C01784=1018.321,266.101,-148.009,-25.446,21.246,-34.279
C01785=1018.328,265.821,-147.958,-25.406,21.239,-34.538
C01786=1018.334,265.575,-147.912,-25.370,21.233,-34.766
C01787=1018.341,265.330,-147.868,-25.335,21.229,-34.991
C01788=1018.347,265.084,-147.824,-25.300,21.225,-35.219
C01789=1018.352,264.837,-147.781,-25.265,21.221,-35.444
C01790=1018.357,264.558,-147.733,-25.226,21.219,-35.699
C01791=1018.363,264.279,-147.684,-25.186,21.217,-35.952
C01792=1018.367,264.000,-147.637,-25.147,21.216,-36.205
C01793=1018.371,263.721,-147.591,-25.108,21.215,-36.458
C01794=1018.374,263.474,-147.551,-25.074,21.216,-36.681
C01795=1018.377,263.227,-147.511,-25.040,21.217,-36.903
C01796=1018.379,262.980,-147.472,-25.006,21.220,-37.124
C01797=1018.382,262.733,-147.433,-24.973,21.223,-37.345
C01798=1018.384,262.453,-147.389,-24.935,21.227,-37.593
C01799=1018.386,262.174,-147.346,-24.897,21.233,-37.842
C01800=1018.387,261.895,-147.304,-24.860,21.238,-38.090
C01801=1018.387,261.616,-147.262,-24.823,21.245,-38.337
C01802=1018.388,261.368,-147.227,-24.790,21.251,-38.554
C01803=1018.388,261.121,-147.191,-24.758,21.259,-38.770
C01804=1018.388,260.874,-147.156,-24.725,21.267,-38.988
C01805=1018.386,260.625,-147.121,-24.693,21.275,-39.204
C01806=1018.385,260.346,-147.083,-24.658,21.287,-39.446
C01807=1018.383,260.066,-147.044,-24.622,21.298,-39.688
C01808=1018.381,259.787,-147.008,-24.587,21.310,-39.930
C01809=1018.378,259.507,-146.971,-24.551,21.322,-40.171
C01810=1018.361,258.272,-146.818,-24.430,21.375,-41.012
C01811=1018.358,258.028,-146.788,-24.430,21.375,-41.014
C01812=1018.355,257.784,-146.759,-24.429,21.375,-41.018
C01813=1018.351,257.541,-146.731,-24.429,21.376,-41.019
C01814=1018.347,257.298,-146.701,-24.429,21.376,-41.021
C01815=1018.344,257.054,-146.671,-24.428,21.375,-41.025
C01816=1018.341,256.811,-146.642,-24.428,21.376,-41.027
C01817=1018.337,256.567,-146.614,-24.428,21.377,-41.029
C01818=1018.334,256.318,-146.584,-24.427,21.376,-41.032
C01819=1018.331,256.071,-146.554,-24.427,21.376,-41.034
C01820=1018.327,255.822,-146.525,-24.426,21.376,-41.037
C01821=1018.323,255.574,-146.495,-24.426,21.377,-41.040
C01822=1018.321,255.326,-146.465,-24.426,21.377,-41.042
C01823=1018.317,255.078,-146.435,-24.425,21.377,-41.045
C01824=1018.314,254.829,-146.406,-24.425,21.377,-41.047
C01825=1018.310,254.581,-146.376,-24.425,21.377,-41.049
C01826=1018.307,254.333,-146.347,-24.424,21.378,-41.052
C01827=1018.303,254.084,-146.318,-24.424,21.378,-41.054
C01828=1018.300,253.837,-146.288,-24.424,21.378,-41.058
C01829=1018.297,253.588,-146.258,-24.423,21.378,-41.060
C01830=1018.293,253.341,-146.229,-24.423,21.378,-41.061
C01831=1018.290,253.092,-146.199,-24.423,21.378,-41.065
C01832=1018.287,252.844,-146.170,-24.422,21.379,-41.067
C01833=1018.283,252.595,-146.140,-24.422,21.379,-41.069
C01834=1018.280,252.347,-146.111,-24.421,21.378,-41.072
C01835=1018.277,252.098,-146.081,-24.421,21.379,-41.074
C01836=1018.274,251.850,-146.053,-24.421,21.380,-41.076
C01837=1018.270,251.602,-146.022,-24.421,21.380,-41.078
C01838=1018.267,251.359,-145.994,-24.420,21.380,-41.082
C01839=1018.264,251.116,-145.965,-24.420,21.380,-41.084
C01840=1018.260,250.872,-145.937,-24.420,21.380,-41.085
C01841=1018.258,250.629,-145.908,-24.419,21.380,-41.089
C01842=1018.255,250.385,-145.879,-24.419,21.380,-41.091
C01843=1018.251,250.142,-145.850,-24.419,21.381,-41.093
C01844=1018.248,249.899,-145.821,-24.418,21.381,-41.095
C01845=1018.244,249.656,-145.793,-24.418,21.381,-41.098
C01846=1018.242,249.408,-145.763,-24.418,21.381,-41.100
C01847=1018.238,249.159,-145.734,-24.417,21.381,-41.102
C01848=1018.235,248.911,-145.705,-24.417,21.381,-41.104
C01849=1018.232,248.663,-145.676,-24.417,21.381,-41.107
C01850=1018.229,248.414,-145.646,-24.416,21.381,-41.109
C01851=1018.226,248.166,-145.617,-24.416,21.382,-41.111
C01852=1018.222,247.918,-145.588,-24.416,21.382,-41.113
C01853=1018.219,247.669,-145.558,-24.415,21.382,-41.117
C01854=1018.216,247.421,-145.529,-24.415,21.382,-41.118
C01855=1018.213,247.173,-145.500,-24.415,21.382,-41.120
C01856=1018.210,246.925,-145.471,-24.414,21.383,-41.122
C01857=1018.207,246.676,-145.441,-24.414,21.382,-41.126
C01858=1018.204,246.428,-145.413,-24.414,21.382,-41.127
C01859=1018.200,246.180,-145.384,-24.413,21.383,-41.129
C01860=1018.198,245.932,-145.354,-24.413,21.384,-41.132
C01861=1018.194,245.683,-145.325,-24.413,21.384,-41.134
C01862=1018.191,245.435,-145.296,-24.412,21.384,-41.137
C01863=1018.188,245.187,-145.267,-24.412,21.384,-41.139
C01864=1018.185,244.939,-145.238,-24.412,21.384,-41.141
C01865=1018.182,244.690,-145.209,-24.412,21.384,-41.143
C01866=1018.179,244.447,-145.181,-24.411,21.384,-41.144
C01867=1018.176,244.204,-145.152,-24.411,21.384,-41.148
C01868=1018.172,243.961,-145.124,-24.411,21.384,-41.150
C01869=1018.170,243.717,-145.095,-24.410,21.384,-41.151
C01870=1018.167,243.474,-145.067,-24.410,21.385,-41.153
C01871=1018.164,243.231,-145.038,-24.410,21.385,-41.155
C01872=1018.161,242.988,-145.010,-24.410,21.385,-41.157
C01873=1018.158,242.745,-144.981,-24.409,21.385,-41.159
C01874=1018.155,242.497,-144.953,-24.409,21.385,-41.162
C01875=1018.153,242.248,-144.924,-24.408,21.385,-41.164
C01876=1018.149,241.999,-144.895,-24.408,21.385,-41.166
C01877=1018.146,241.751,-144.866,-24.408,21.386,-41.168
C01878=1018.143,241.503,-144.837,-24.408,21.386,-41.170
C01879=1018.140,241.255,-144.808,-24.407,21.386,-41.172
C01880=1018.138,241.006,-144.779,-24.407,21.386,-41.174
C01881=1018.134,240.758,-144.751,-24.407,21.386,-41.177
C01882=1018.132,240.510,-144.721,-24.406,21.386,-41.179
C01883=1018.129,240.262,-144.692,-24.406,21.386,-41.181
C01884=1018.126,240.013,-144.664,-24.406,21.386,-41.183
C01885=1018.123,239.765,-144.635,-24.406,21.387,-41.184
C01886=1018.120,239.517,-144.606,-24.405,21.387,-41.186
C01887=1018.117,239.268,-144.578,-24.405,21.387,-41.188
C01888=1018.114,239.020,-144.549,-24.405,21.387,-41.190
C01889=1018.111,238.772,-144.520,-24.405,21.388,-41.192
C01890=1018.109,238.523,-144.491,-24.404,21.387,-41.195
C01891=1018.106,238.275,-144.462,-24.404,21.387,-41.197
C01892=1018.102,238.027,-144.434,-24.403,21.388,-41.199
C01893=1018.100,237.778,-144.405,-24.403,21.388,-41.201
C01894=1018.096,237.535,-144.376,-24.403,21.388,-41.203
C01895=1018.094,237.291,-144.348,-24.403,21.388,-41.205
C01896=1018.091,237.049,-144.320,-24.402,21.388,-41.207
C01897=1018.088,236.806,-144.292,-24.402,21.389,-41.209
C01898=1018.086,236.562,-144.264,-24.402,21.389,-41.210
C01899=1018.083,236.320,-144.236,-24.402,21.389,-41.212
C01900=1018.081,236.077,-144.208,-24.401,21.389,-41.214
C01901=1018.078,235.833,-144.181,-24.401,21.390,-41.216
C01902=1018.075,235.585,-144.151,-24.401,21.389,-41.218
C01903=1018.072,235.336,-144.123,-24.401,21.389,-41.219
C01904=1018.069,235.089,-144.094,-24.400,21.389,-41.221
C01905=1018.067,234.840,-144.066,-24.400,21.390,-41.223
C01906=1018.064,234.592,-144.037,-24.400,21.390,-41.225
C01907=1018.061,234.343,-144.009,-24.400,21.390,-41.227
C01908=1018.058,234.095,-143.980,-24.399,21.390,-41.229
C01909=1018.055,233.846,-143.951,-24.399,21.390,-41.231
C01910=1018.053,233.598,-143.922,-24.399,21.391,-41.233
C01911=1018.050,233.350,-143.894,-24.399,21.391,-41.234
C01912=1018.047,233.101,-143.866,-24.398,21.391,-41.236
C01913=1018.045,232.853,-143.837,-24.398,21.390,-41.238
C01914=1018.042,232.605,-143.809,-24.398,21.391,-41.240
C01915=1018.039,232.357,-143.780,-24.397,21.391,-41.242
C01916=1018.036,232.108,-143.751,-24.397,21.391,-41.243
C01917=1018.034,231.860,-143.724,-24.397,21.391,-41.245
C01918=1018.031,231.612,-143.694,-24.397,21.392,-41.247
C01919=1018.028,231.363,-143.666,-24.396,21.392,-41.249
C01920=1018.026,231.114,-143.638,-24.396,21.392,-41.251
C01921=1018.023,230.866,-143.609,-24.396,21.391,-41.252
C01922=1018.021,230.624,-143.582,-24.396,21.392,-41.254
C01923=1018.018,230.380,-143.554,-24.395,21.392,-41.256
C01924=1018.015,230.137,-143.526,-24.395,21.392,-41.258
C01925=1018.013,229.894,-143.499,-24.395,21.392,-41.260
C01926=1018.010,229.652,-143.470,-24.395,21.392,-41.262
C01927=1018.008,229.408,-143.442,-24.394,21.392,-41.263
C01928=1018.005,229.166,-143.415,-24.394,21.392,-41.265
C01929=1018.002,228.922,-143.388,-24.394,21.393,-41.266
C01930=1018.000,228.673,-143.359,-24.394,21.393,-41.267
C01931=1017.997,228.426,-143.331,-24.394,21.393,-41.269
C01932=1017.995,228.177,-143.302,-24.393,21.394,-41.271
C01933=1017.992,227.929,-143.274,-24.393,21.393,-41.273
C01934=1017.990,227.681,-143.246,-24.393,21.393,-41.275
C01935=1017.988,227.432,-143.217,-24.393,21.393,-41.276
C01936=1017.985,227.183,-143.189,-24.392,21.394,-41.278
C01937=1017.981,226.935,-143.161,-24.392,21.394,-41.280
C01938=1017.980,226.687,-143.132,-24.392,21.393,-41.282
C01939=1017.977,226.439,-143.104,-24.391,21.393,-41.284
C01940=1017.975,226.190,-143.076,-24.391,21.394,-41.285
C01941=1017.972,225.942,-143.048,-24.391,21.395,-41.286
C01942=1017.969,225.693,-143.020,-24.391,21.395,-41.288
C01943=1017.968,225.445,-142.992,-24.391,21.394,-41.289
C01944=1017.965,225.196,-142.963,-24.390,21.394,-41.291
C01945=1017.962,224.948,-142.935,-24.390,21.395,-41.293
C01946=1017.960,224.700,-142.907,-24.390,21.395,-41.295
C01947=1017.957,224.452,-142.878,-24.390,21.395,-41.297
C01948=1017.954,224.204,-142.851,-24.389,21.394,-41.298
C01949=1017.952,223.955,-142.822,-24.389,21.395,-41.300
C01950=1017.949,223.695,-142.793,-24.389,21.395,-41.300
C01951=1017.948,223.437,-142.764,-24.389,21.396,-41.302
C01952=1017.945,223.177,-142.734,-24.389,21.396,-41.304
C01953=1017.942,222.918,-142.705,-24.388,21.396,-41.306
C01954=1017.940,222.670,-142.677,-24.388,21.395,-41.308
C01955=1017.937,222.421,-142.649,-24.388,21.396,-41.309
C01956=1017.936,222.173,-142.621,-24.388,21.396,-41.311
C01957=1017.933,221.924,-142.593,-24.387,21.396,-41.313
C01958=1017.930,221.676,-142.565,-24.387,21.395,-41.315
C01959=1017.928,221.428,-142.536,-24.387,21.396,-41.315
C01960=1017.925,221.179,-142.508,-24.387,21.397,-41.317
C01961=1017.923,220.931,-142.481,-24.387,21.397,-41.319
C01962=1017.921,220.682,-142.452,-24.386,21.396,-41.320
C01963=1017.918,220.434,-142.424,-24.386,21.396,-41.322
C01964=1017.915,220.186,-142.396,-24.386,21.397,-41.324
C01965=1017.914,219.937,-142.369,-24.386,21.397,-41.325
C01966=1017.912,219.689,-142.341,-24.385,21.397,-41.326
C01967=1017.909,219.440,-142.313,-24.385,21.397,-41.328
C01968=1017.907,219.192,-142.284,-24.385,21.397,-41.330
C01969=1017.904,218.944,-142.256,-24.385,21.397,-41.332
C01970=1017.902,218.695,-142.228,-24.384,21.397,-41.333
C01971=1017.900,218.446,-142.201,-24.384,21.398,-41.333
C01972=1017.897,218.198,-142.173,-24.384,21.398,-41.335
C01973=1017.895,217.949,-142.144,-24.384,21.398,-41.337
C01974=1017.893,217.724,-142.119,-24.384,21.397,-41.339
C01975=1017.891,217.497,-142.094,-24.383,21.398,-41.341
C01976=1017.889,217.270,-142.068,-24.383,21.399,-41.341
C01977=1017.887,217.043,-142.044,-24.383,21.398,-41.342
C01978=1017.885,216.800,-142.016,-24.383,21.398,-41.344
C01979=1017.883,216.558,-141.989,-24.383,21.398,-41.346
C01980=1017.881,216.315,-141.961,-24.383,21.398,-41.346
C01981=1017.878,216.072,-141.934,-24.382,21.399,-41.348
C01982=1017.876,215.829,-141.907,-24.382,21.399,-41.350
C01983=1017.874,215.586,-141.880,-24.382,21.399,-41.352
C01984=1017.872,215.343,-141.852,-24.382,21.398,-41.353
C01985=1017.869,215.101,-141.825,-24.382,21.399,-41.354
C01986=1017.868,214.852,-141.798,-24.381,21.400,-41.356
C01987=1017.865,214.604,-141.770,-24.381,21.399,-41.357
C01988=1017.863,214.356,-141.742,-24.381,21.399,-41.359
C01989=1017.861,214.107,-141.714,-24.381,21.400,-41.359
C01990=1017.859,213.859,-141.687,-24.381,21.400,-41.361
C01991=1017.857,213.610,-141.658,-24.380,21.400,-41.363
C01992=1017.855,213.362,-141.631,-24.380,21.400,-41.365
C01993=1017.852,213.114,-141.603,-24.380,21.400,-41.366
C01994=1017.851,212.865,-141.576,-24.380,21.400,-41.366
C01995=1017.848,212.616,-141.548,-24.380,21.400,-41.368
C01996=1017.846,212.368,-141.520,-24.379,21.400,-41.370
C01997=1017.844,212.120,-141.492,-24.379,21.400,-41.372
C01998=1017.841,211.871,-141.464,-24.379,21.401,-41.372
C01999=1017.839,211.622,-141.437,-24.379,21.401,-41.374
C02000=1017.838,211.374,-141.409,-24.378,21.400,-41.375
C02001=1017.836,211.126,-141.382,-24.378,21.400,-41.377
C02002=1017.833,210.878,-141.354,-24.378,21.401,-41.378
C02003=1017.831,210.628,-141.326,-24.378,21.401,-41.379
C02004=1017.829,210.380,-141.299,-24.378,21.401,-41.381
C02005=1017.828,210.132,-141.271,-24.377,21.401,-41.383
C02006=1017.825,209.889,-141.244,-24.377,21.401,-41.383
C02007=1017.823,209.647,-141.217,-24.377,21.401,-41.385
C02008=1017.822,209.404,-141.191,-24.377,21.402,-41.387
C02009=1017.819,209.162,-141.163,-24.377,21.401,-41.388
C02010=1017.818,208.918,-141.136,-24.377,21.402,-41.389
C02011=1017.815,208.676,-141.109,-24.376,21.402,-41.391
C02012=1017.813,208.433,-141.082,-24.376,21.401,-41.392
C02013=1017.812,208.191,-141.056,-24.376,21.402,-41.392
C02014=1017.809,207.942,-141.028,-24.376,21.402,-41.394
C02015=1017.807,207.693,-141.000,-24.376,21.402,-41.396
C02016=1017.805,207.445,-140.973,-24.375,21.402,-41.398
C02017=1017.804,207.197,-140.945,-24.375,21.402,-41.398
C02018=1017.802,206.948,-140.918,-24.375,21.402,-41.399
C02019=1017.799,206.700,-140.890,-24.375,21.402,-41.401
C02020=1017.798,206.451,-140.863,-24.375,21.402,-41.401
C02021=1017.796,206.203,-140.836,-24.375,21.403,-41.403
C02022=1017.794,205.955,-140.808,-24.374,21.403,-41.405
C02023=1017.792,205.705,-140.780,-24.374,21.402,-41.407
C02024=1017.790,205.457,-140.753,-24.374,21.403,-41.407
C02025=1017.788,205.209,-140.725,-24.374,21.403,-41.409
C02026=1017.786,204.960,-140.698,-24.373,21.403,-41.410
C02027=1017.784,204.712,-140.671,-24.374,21.404,-41.411
C02028=1017.783,204.463,-140.643,-24.373,21.403,-41.412
C02029=1017.780,204.215,-140.615,-24.373,21.403,-41.414
C02030=1017.778,203.966,-140.589,-24.373,21.404,-41.415
C02031=1017.777,203.718,-140.561,-24.373,21.403,-41.416
C02032=1017.771,202.502,-140.425,-24.425,21.378,-41.051
C02033=1017.769,202.114,-140.381,-24.424,21.378,-41.052
C02034=1017.768,201.765,-140.342,-24.424,21.378,-41.054
C02035=1017.769,201.414,-140.303,-24.424,21.378,-41.058
C02036=1017.769,201.006,-140.259,-24.423,21.379,-41.060
C02037=1017.770,200.779,-140.234,-24.423,21.378,-41.061
C02038=1017.771,200.550,-140.209,-24.423,21.378,-41.063
C02039=1017.771,200.327,-140.184,-24.423,21.378,-41.065
C02040=1017.771,200.115,-140.161,-24.423,21.378,-41.065
C02041=1017.772,199.714,-140.117,-24.422,21.379,-41.069
C02042=1017.772,199.325,-140.074,-24.422,21.379,-41.071
C02043=1017.773,198.926,-140.031,-24.421,21.379,-41.074
C02044=1017.773,198.525,-139.988,-24.421,21.379,-41.076
C02045=1017.774,198.125,-139.944,-24.421,21.380,-41.078
C02046=1017.775,197.723,-139.900,-24.420,21.380,-41.082
C02047=1017.776,197.322,-139.856,-24.420,21.380,-41.084
C02048=1017.776,196.921,-139.812,-24.419,21.380,-41.087
C02049=1017.777,196.519,-139.769,-24.419,21.380,-41.089
C02050=1017.777,196.119,-139.725,-24.419,21.381,-41.091
C02051=1017.779,195.717,-139.681,-24.418,21.380,-41.094
C02052=1017.779,195.317,-139.637,-24.418,21.381,-41.097
C02053=1017.780,194.915,-139.593,-24.418,21.381,-41.100
C02054=1017.781,194.514,-139.550,-24.417,21.381,-41.102
C02055=1017.781,194.113,-139.507,-24.417,21.381,-41.105
C02056=1017.783,193.712,-139.462,-24.417,21.382,-41.108
C02057=1017.783,193.311,-139.419,-24.416,21.382,-41.109
C02058=1017.784,192.910,-139.375,-24.416,21.382,-41.113
C02059=1017.785,192.508,-139.332,-24.415,21.382,-41.115
C02060=1017.785,192.108,-139.288,-24.415,21.382,-41.118
C02061=1017.786,191.707,-139.245,-24.415,21.382,-41.120
C02062=1017.787,191.305,-139.202,-24.414,21.382,-41.124
C02063=1017.788,190.904,-139.158,-24.414,21.383,-41.126
C02064=1017.789,190.503,-139.114,-24.414,21.383,-41.128
C02065=1017.789,190.102,-139.070,-24.413,21.383,-41.131
C02066=1017.790,189.701,-139.027,-24.413,21.383,-41.133
C02067=1017.791,189.300,-138.984,-24.412,21.384,-41.137
C02068=1017.792,188.899,-138.941,-24.412,21.384,-41.139
C02069=1017.793,188.498,-138.897,-24.412,21.384,-41.141
C02070=1017.794,188.097,-138.854,-24.411,21.384,-41.144
C02071=1017.794,187.695,-138.811,-24.411,21.385,-41.146
C02072=1017.796,187.295,-138.768,-24.411,21.384,-41.150
C02073=1017.797,186.894,-138.724,-24.410,21.384,-41.151
C02074=1017.797,186.493,-138.681,-24.410,21.384,-41.155
C02075=1017.798,186.091,-138.638,-24.410,21.385,-41.157
C02076=1017.800,185.691,-138.594,-24.409,21.385,-41.159
C02077=1017.801,185.289,-138.551,-24.409,21.385,-41.162
C02078=1017.802,184.889,-138.508,-24.409,21.386,-41.165
C02079=1017.803,184.488,-138.465,-24.408,21.386,-41.168
C02080=1017.804,184.086,-138.421,-24.408,21.386,-41.170
C02081=1017.804,183.686,-138.379,-24.407,21.386,-41.172
C02082=1017.805,183.285,-138.336,-24.407,21.386,-41.176
C02083=1017.806,182.884,-138.293,-24.407,21.387,-41.177
C02084=1017.808,182.483,-138.250,-24.406,21.386,-41.181
C02085=1017.809,182.082,-138.207,-24.406,21.387,-41.183
C02086=1017.810,181.681,-138.164,-24.405,21.387,-41.186
C02087=1017.811,181.280,-138.121,-24.405,21.387,-41.188
C02088=1017.812,180.879,-138.078,-24.405,21.387,-41.190
C02089=1017.813,180.479,-138.035,-24.404,21.388,-41.194
C02090=1017.814,180.078,-137.992,-24.404,21.388,-41.196
C02091=1017.815,179.676,-137.949,-24.403,21.388,-41.199
C02092=1017.817,179.276,-137.906,-24.403,21.388,-41.201
C02093=1017.818,178.875,-137.863,-24.403,21.388,-41.205
C02094=1017.818,178.474,-137.821,-24.402,21.388,-41.207
C02095=1017.820,178.074,-137.778,-24.402,21.389,-41.209
C02096=1017.821,177.673,-137.735,-24.402,21.389,-41.212
C02097=1017.822,177.272,-137.692,-24.401,21.389,-41.214
C02098=1017.823,176.871,-137.649,-24.401,21.389,-41.218
C02099=1017.825,176.471,-137.606,-24.401,21.389,-41.219
C02100=1017.826,176.070,-137.565,-24.400,21.390,-41.223
C02101=1017.827,175.669,-137.522,-24.400,21.390,-41.225
C02102=1017.828,175.269,-137.479,-24.400,21.390,-41.227
C02103=1017.829,174.867,-137.436,-24.399,21.390,-41.231
C02104=1017.830,174.467,-137.394,-24.399,21.391,-41.233
C02105=1017.831,174.066,-137.351,-24.398,21.390,-41.236
C02106=1017.833,173.665,-137.309,-24.398,21.390,-41.238
C02107=1017.834,173.265,-137.266,-24.397,21.391,-41.242
C02108=1017.835,172.864,-137.223,-24.397,21.391,-41.243
C02109=1017.837,172.463,-137.181,-24.397,21.391,-41.247
C02110=1017.838,172.063,-137.138,-24.396,21.392,-41.249
C02111=1017.838,171.663,-137.096,-24.396,21.392,-41.251
C02112=1017.840,171.261,-137.053,-24.396,21.392,-41.254
C02113=1017.841,170.861,-137.010,-24.395,21.392,-41.256
C02114=1017.842,170.461,-136.968,-24.395,21.392,-41.260
C02115=1017.844,170.060,-136.926,-24.395,21.392,-41.262
C02116=1017.845,169.660,-136.884,-24.394,21.392,-41.265
C02117=1017.846,169.475,-136.864,-24.394,21.393,-41.266
C02118=1017.847,169.074,-136.821,-24.394,21.392,-41.269
C02119=1017.848,168.858,-136.799,-24.393,21.393,-41.271
C02120=1017.849,168.458,-136.756,-24.393,21.393,-41.273
C02121=1017.851,168.058,-136.715,-24.393,21.394,-41.275
C02122=1017.851,167.658,-136.672,-24.392,21.394,-41.278
C02123=1017.853,167.257,-136.630,-24.392,21.394,-41.280
C02124=1017.854,166.856,-136.588,-24.391,21.393,-41.284
C02125=1017.856,166.456,-136.546,-24.391,21.395,-41.286
C02126=1017.857,166.056,-136.503,-24.391,21.394,-41.289
C02127=1017.858,165.655,-136.460,-24.390,21.394,-41.291
C02128=1017.859,165.255,-136.419,-24.390,21.395,-41.295
C02129=1017.861,164.855,-136.376,-24.390,21.395,-41.297
C02130=1017.862,164.455,-136.335,-24.389,21.395,-41.300
C02131=1017.863,164.069,-136.294,-24.389,21.395,-41.302
C02132=1017.864,163.879,-136.274,-24.389,21.395,-41.304
C02133=1017.865,163.467,-136.231,-24.388,21.396,-41.306
C02134=1017.866,163.231,-136.206,-24.388,21.395,-41.308
C02135=1017.867,162.977,-136.179,-24.388,21.396,-41.309
C02136=1017.869,162.714,-136.152,-24.388,21.396,-41.311
C02137=1017.869,162.446,-136.123,-24.387,21.396,-41.313
C02138=1017.870,162.174,-136.096,-24.387,21.396,-41.315
C02139=1017.871,161.905,-136.067,-24.387,21.397,-41.317
C02140=1017.872,161.642,-136.039,-24.387,21.397,-41.319
C02141=1017.872,161.391,-136.013,-24.386,21.396,-41.320
C02142=1017.873,161.154,-135.988,-24.386,21.396,-41.322
C02143=1017.874,160.929,-135.965,-24.386,21.397,-41.324
C02144=1017.875,160.716,-135.943,-24.386,21.397,-41.325
C02145=1017.877,160.311,-135.900,-24.385,21.397,-41.328
C02146=1017.878,159.914,-135.858,-24.385,21.397,-41.330
C02147=1017.880,159.514,-135.817,-24.384,21.398,-41.333
C02148=1017.887,159.113,-135.778,-24.384,21.398,-41.335
C02149=1017.893,158.713,-135.739,-24.384,21.397,-41.339
C02150=1017.900,158.242,-135.694,-24.383,21.398,-41.342
C02151=1017.905,157.908,-135.661,-24.383,21.398,-41.344
C02152=1017.911,157.504,-135.622,-24.383,21.398,-41.346
C02153=1017.918,157.100,-135.583,-24.382,21.399,-41.350
C02154=1017.925,156.695,-135.543,-24.382,21.399,-41.352
C02155=1017.931,156.288,-135.504,-24.381,21.399,-41.355
C02156=1017.936,155.882,-135.465,-24.381,21.400,-41.358
C02157=1017.943,155.474,-135.425,-24.381,21.399,-41.361
C02158=1017.949,155.066,-135.386,-24.380,21.400,-41.363
C02159=1017.956,154.657,-135.346,-24.380,21.400,-41.366
C02160=1017.962,154.247,-135.306,-24.380,21.400,-41.368
C02161=1017.969,153.836,-135.266,-24.379,21.401,-41.372
C02162=1017.975,153.424,-135.227,-24.378,21.400,-41.375
C02163=1017.980,153.013,-135.186,-24.378,21.400,-41.377
C02164=1017.987,152.601,-135.146,-24.378,21.401,-41.381
C02165=1017.993,152.188,-135.107,-24.377,21.401,-41.383
C02166=1017.999,151.775,-135.067,-24.377,21.402,-41.387
C02167=1018.005,151.361,-135.027,-24.377,21.402,-41.389
C02168=1018.012,150.948,-134.987,-24.376,21.401,-41.392
C02169=1018.018,150.534,-134.947,-24.376,21.402,-41.394
C02170=1018.024,150.120,-134.907,-24.375,21.402,-41.398
C02171=1018.030,149.706,-134.867,-24.375,21.402,-41.401
C02172=1018.036,149.292,-134.827,-24.375,21.403,-41.403
C02173=1018.042,148.878,-134.787,-24.374,21.403,-41.407
C02174=1018.048,148.464,-134.747,-24.374,21.403,-41.409
C02175=1018.054,148.050,-134.707,-24.373,21.403,-41.412
C02176=1018.060,147.636,-134.667,-24.373,21.403,-41.416
C02177=1018.066,147.223,-134.626,-24.372,21.404,-41.418
C02178=1018.073,146.809,-134.586,-24.372,21.404,-41.422
C02179=1018.078,146.395,-134.547,-24.372,21.404,-41.424
C02180=1018.084,145.983,-134.506,-24.371,21.405,-41.427
C02181=1018.090,145.571,-134.467,-24.371,21.404,-41.431
C02182=1018.096,145.158,-134.427,-24.370,21.405,-41.432
C02183=1018.102,144.747,-134.388,-24.370,21.405,-41.436
C02184=1018.108,144.336,-134.348,-24.370,21.405,-41.438
C02185=1018.114,143.926,-134.308,-24.369,21.406,-41.442
C02186=1018.120,143.516,-134.268,-24.369,21.405,-41.445
C02187=1018.125,143.107,-134.229,-24.368,21.406,-41.448
C02188=1018.131,142.699,-134.190,-24.368,21.406,-41.451
C02189=1018.137,142.292,-134.150,-24.368,21.406,-41.453
C02190=1018.143,141.886,-134.111,-24.367,21.407,-41.457
C02191=1018.148,141.481,-134.072,-24.366,21.406,-41.460
C02192=1018.154,141.076,-134.034,-24.366,21.407,-41.462
C02193=1018.160,140.659,-133.994,-24.366,21.408,-41.466
C02194=1018.163,140.423,-133.970,-24.366,21.408,-41.468
C02195=1018.167,140.164,-133.945,-24.365,21.408,-41.470
C02196=1018.171,139.887,-133.919,-24.365,21.408,-41.471
C02197=1018.174,139.599,-133.891,-24.365,21.408,-41.473
C02198=1018.179,139.312,-133.863,-24.364,21.408,-41.475
C02199=1018.182,139.034,-133.836,-24.364,21.407,-41.476
C02200=1018.186,138.774,-133.811,-24.364,21.408,-41.478
C02201=1018.189,138.536,-133.788,-24.364,21.408,-41.480
C02202=1018.192,138.320,-133.768,-24.363,21.408,-41.482
C02203=1018.195,138.114,-133.748,-24.363,21.408,-41.484
C02204=1018.200,137.713,-133.709,-24.363,21.408,-41.486
C02205=1018.206,137.343,-133.674,-24.363,21.410,-41.488
C02206=1018.210,137.006,-133.641,-24.362,21.409,-41.491
C02207=1018.214,136.690,-133.610,-24.361,21.409,-41.495
C02208=1018.219,136.372,-133.580,-24.361,21.410,-41.497
C02209=1018.223,136.033,-133.547,-24.361,21.409,-41.500
C02210=1018.228,135.661,-133.512,-24.360,21.410,-41.502
C02211=1018.233,135.266,-133.474,-24.360,21.411,-41.505
C02212=1018.238,134.867,-133.435,-24.360,21.410,-41.508
C02213=1018.244,134.469,-133.397,-24.359,21.411,-41.510
C02214=1018.249,134.070,-133.359,-24.359,21.411,-41.514
C02215=1018.254,133.671,-133.320,-24.358,21.411,-41.517
C02216=1018.260,133.272,-133.283,-24.358,21.412,-41.519
C02217=1018.265,132.874,-133.244,-24.358,21.411,-41.523
C02218=1018.270,132.475,-133.205,-24.357,21.412,-41.525
C02219=1018.276,132.076,-133.167,-24.357,21.412,-41.528
C02220=1018.280,131.678,-133.129,-24.356,21.412,-41.532
C02221=1018.286,131.278,-133.091,-24.356,21.413,-41.534
C02222=1018.291,130.880,-133.053,-24.356,21.413,-41.538
C02223=1018.296,130.482,-133.014,-24.355,21.413,-41.541
C02224=1018.301,130.083,-132.976,-24.355,21.413,-41.543
C02225=1018.306,129.685,-132.938,-24.354,21.413,-41.547
C02226=1018.312,129.286,-132.899,-24.354,21.413,-41.550
C02227=1018.316,128.887,-132.862,-24.354,21.414,-41.552
C02228=1018.322,128.489,-132.824,-24.353,21.414,-41.555
C02229=1018.327,128.090,-132.785,-24.353,21.415,-41.558
C02230=1018.332,127.691,-132.747,-24.352,21.414,-41.561
C02231=1018.337,127.293,-132.709,-24.352,21.415,-41.565
C02232=1018.342,126.894,-132.670,-24.351,21.415,-41.567
C02233=1018.347,126.495,-132.632,-24.351,21.415,-41.571
C02234=1018.351,126.097,-132.594,-24.350,21.415,-41.574
C02235=1018.356,125.699,-132.556,-24.350,21.416,-41.576
C02236=1018.361,125.300,-132.518,-24.350,21.416,-41.580
C02237=1018.367,124.901,-132.479,-24.349,21.416,-41.583
C02238=1018.372,124.503,-132.441,-24.349,21.416,-41.585
C02239=1018.377,124.104,-132.404,-24.348,21.417,-41.589
C02240=1018.381,123.705,-132.365,-24.348,21.416,-41.592
C02241=1018.386,123.308,-132.327,-24.348,21.418,-41.595
C02242=1018.391,122.909,-132.290,-24.347,21.417,-41.598
C02243=1018.396,122.510,-132.251,-24.347,21.418,-41.602
C02244=1018.400,122.112,-132.213,-24.346,21.417,-41.605
C02245=1018.406,121.713,-132.176,-24.346,21.418,-41.607
C02246=1018.411,121.314,-132.137,-24.345,21.418,-41.611
C02247=1018.415,120.916,-132.098,-24.345,21.418,-41.614
C02248=1018.420,120.517,-132.061,-24.345,21.419,-41.617
C02249=1018.425,120.119,-132.023,-24.344,21.419,-41.620
C02250=1018.430,119.720,-131.985,-24.343,21.419,-41.624
C02251=1018.435,119.322,-131.947,-24.343,21.420,-41.626
C02252=1018.440,118.923,-131.909,-24.343,21.420,-41.629
C02253=1018.445,118.525,-131.871,-24.342,21.420,-41.633
C02254=1018.451,118.127,-131.834,-24.342,21.420,-41.637
C02255=1018.455,117.727,-131.796,-24.341,21.420,-41.638
C02256=1018.461,117.330,-131.758,-24.341,21.421,-41.642
C02257=1018.465,116.930,-131.721,-24.340,21.420,-41.646
C02258=1018.471,116.533,-131.683,-24.340,21.421,-41.649
C02259=1018.475,116.133,-131.645,-24.340,21.422,-41.652
C02260=1018.481,115.735,-131.608,-24.339,21.422,-41.655
C02261=1018.485,115.337,-131.569,-24.339,21.422,-41.659
C02262=1018.489,114.938,-131.532,-24.338,21.422,-41.662
C02263=1018.495,114.540,-131.494,-24.338,21.423,-41.664
C02264=1018.499,114.141,-131.456,-24.337,21.422,-41.668
C02265=1018.505,113.742,-131.419,-24.337,21.423,-41.671
C02266=1018.509,113.344,-131.381,-24.336,21.423,-41.675
C02267=1018.515,112.945,-131.344,-24.336,21.423,-41.677
C02268=1018.519,112.547,-131.306,-24.335,21.424,-41.681
C02269=1018.524,112.149,-131.268,-24.335,21.423,-41.684
C02270=1018.529,111.750,-131.231,-24.334,21.424,-41.688
C02271=1018.533,111.351,-131.192,-24.334,21.425,-41.690
C02272=1018.539,110.953,-131.155,-24.334,21.425,-41.694
C02273=1018.543,110.554,-131.118,-24.333,21.425,-41.697
C02274=1018.547,110.155,-131.080,-24.333,21.425,-41.701
C02275=1018.553,109.757,-131.042,-24.332,21.426,-41.703
C02276=1018.557,109.358,-131.005,-24.332,21.426,-41.707
C02277=1018.562,108.960,-130.967,-24.331,21.426,-41.710
C02278=1018.567,108.561,-130.930,-24.331,21.426,-41.714
C02279=1018.571,108.162,-130.893,-24.330,21.426,-41.717
C02280=1018.576,107.764,-130.854,-24.330,21.427,-41.719
C02281=1018.581,107.365,-130.817,-24.330,21.427,-41.723
C02282=1018.585,106.967,-130.780,-24.329,21.427,-41.727
C02283=1018.590,106.568,-130.742,-24.328,21.427,-41.730
C02284=1018.594,106.170,-130.705,-24.328,21.428,-41.734
C02285=1018.599,105.771,-130.667,-24.328,21.428,-41.736
C02286=1018.603,105.372,-130.630,-24.327,21.429,-41.740
C02287=1018.608,104.973,-130.592,-24.327,21.429,-41.743
C02288=1018.613,104.574,-130.554,-24.326,21.429,-41.747
C02289=1018.617,104.176,-130.517,-24.326,21.429,-41.751
C02290=1018.622,103.778,-130.479,-24.325,21.430,-41.754
C02291=1018.626,103.379,-130.442,-24.325,21.430,-41.756
C02292=1018.630,102.980,-130.405,-24.324,21.430,-41.760
C02293=1018.635,102.581,-130.367,-24.324,21.430,-41.763
C02294=1018.639,102.182,-130.330,-24.323,21.430,-41.767
C02295=1018.644,101.784,-130.292,-24.323,21.431,-41.771
C02296=1018.648,101.385,-130.255,-24.322,21.431,-41.775
C02297=1018.653,100.986,-130.217,-24.322,21.431,-41.778
C02298=1018.657,100.588,-130.180,-24.322,21.432,-41.780
C02299=1018.661,100.189,-130.143,-24.321,21.432,-41.784
C02300=1018.666,99.790,-130.105,-24.320,21.432,-41.787
C02301=1018.670,99.391,-130.068,-24.320,21.432,-41.791
C02302=1018.675,98.992,-130.030,-24.319,21.433,-41.795
C02303=1018.679,98.593,-129.993,-24.319,21.432,-41.798
C02304=1018.683,98.195,-129.956,-24.318,21.433,-41.802
C02305=1018.687,97.796,-129.919,-24.318,21.433,-41.806
C02306=1018.692,97.397,-129.881,-24.318,21.434,-41.808
C02307=1018.696,96.998,-129.844,-24.317,21.434,-41.811
C02308=1018.700,96.600,-129.807,-24.317,21.435,-41.815
C02309=1018.705,96.200,-129.769,-24.316,21.435,-41.819
C02310=1018.708,95.801,-129.731,-24.316,21.435,-41.822
C02311=1018.712,95.402,-129.694,-24.315,21.435,-41.826
C02312=1018.716,95.003,-129.657,-24.315,21.436,-41.830
C02313=1018.721,94.604,-129.620,-24.314,21.435,-41.833
C02314=1018.725,94.205,-129.583,-24.313,21.436,-41.837
C02315=1018.729,93.806,-129.546,-24.313,21.436,-41.841
C02316=1018.733,93.407,-129.508,-24.312,21.437,-41.844
C02317=1018.737,93.008,-129.471,-24.312,21.437,-41.846
C02318=1018.741,92.609,-129.434,-24.312,21.437,-41.850
C02319=1018.746,92.210,-129.396,-24.311,21.438,-41.854
C02320=1018.749,91.811,-129.359,-24.311,21.438,-41.857
C02321=1018.753,91.412,-129.322,-24.310,21.438,-41.861
C02322=1018.758,91.012,-129.285,-24.310,21.438,-41.865
C02323=1018.761,90.613,-129.248,-24.309,21.439,-41.868
C02324=1018.765,90.214,-129.211,-24.309,21.439,-41.872
C02325=1018.769,89.816,-129.173,-24.308,21.439,-41.875
C02326=1018.773,89.422,-129.137,-24.308,21.439,-41.879
C02327=1018.777,89.036,-129.101,-24.307,21.440,-41.883
C02328=1018.781,88.653,-129.065,-24.307,21.440,-41.887
C02329=1018.785,88.270,-129.030,-24.306,21.440,-41.890
C02330=1018.789,87.882,-128.993,-24.305,21.440,-41.894
C02331=1018.793,87.485,-128.957,-24.305,21.441,-41.898
C02332=1018.796,87.083,-128.920,-24.304,21.441,-41.901
C02333=1018.800,86.677,-128.882,-24.304,21.442,-41.905
C02334=1018.804,86.270,-128.844,-24.303,21.441,-41.908
C02335=1018.808,85.860,-128.806,-24.303,21.442,-41.912
C02336=1018.812,85.449,-128.768,-24.302,21.442,-41.916
C02337=1018.815,85.037,-128.729,-24.302,21.443,-41.920
C02338=1018.820,84.623,-128.691,-24.301,21.443,-41.923
C02339=1018.824,84.207,-128.653,-24.301,21.443,-41.927
C02340=1018.827,83.790,-128.614,-24.300,21.444,-41.931
C02341=1018.832,83.371,-128.575,-24.300,21.444,-41.935
C02342=1018.835,82.951,-128.536,-24.299,21.444,-41.938
C02343=1018.837,82.740,-128.517,-24.299,21.444,-41.940
C02344=1018.840,82.529,-128.497,-24.299,21.444,-41.942
C02345=1018.841,82.319,-128.478,-24.299,21.445,-41.944
C02346=1018.843,82.106,-128.458,-24.298,21.444,-41.947
C02347=1018.845,81.895,-128.439,-24.298,21.445,-41.949
C02348=1018.847,81.683,-128.419,-24.298,21.445,-41.951
C02349=1018.849,81.471,-128.399,-24.297,21.445,-41.953
C02350=1018.850,81.258,-128.380,-24.297,21.445,-41.955
C02351=1018.853,81.046,-128.360,-24.297,21.445,-41.956
C02352=1018.855,80.833,-128.340,-24.297,21.446,-41.958
C02353=1018.857,80.620,-128.320,-24.296,21.446,-41.960
C02354=1018.859,80.407,-128.300,-24.296,21.446,-41.962
C02355=1018.861,80.196,-128.282,-24.296,21.446,-41.964
C02356=1018.863,79.986,-128.262,-24.296,21.447,-41.966
C02357=1018.866,79.571,-128.224,-24.295,21.447,-41.970
C02358=1018.870,79.165,-128.187,-24.294,21.447,-41.973
C02359=1018.873,78.768,-128.150,-24.294,21.447,-41.977
C02360=1018.877,78.378,-128.113,-24.293,21.448,-41.980
C02361=1018.880,77.991,-128.079,-24.293,21.447,-41.986
C02362=1018.884,77.605,-128.042,-24.292,21.448,-41.989
C02363=1018.887,77.216,-128.007,-24.292,21.449,-41.994
C02364=1018.890,76.822,-127.970,-24.291,21.449,-41.997
C02365=1018.894,76.419,-127.933,-24.291,21.449,-42.001
C02366=1018.898,76.008,-127.895,-24.290,21.450,-42.004
C02367=1018.901,75.589,-127.856,-24.290,21.450,-42.008
C02368=1018.903,75.376,-127.837,-24.289,21.451,-42.010
C02369=1018.906,75.162,-127.818,-24.289,21.451,-42.012
C02370=1018.906,74.949,-127.797,-24.289,21.450,-42.015
C02371=1018.909,74.735,-127.778,-24.288,21.451,-42.017
C02372=1018.910,74.522,-127.758,-24.288,21.451,-42.019
C02373=1018.912,74.309,-127.739,-24.288,21.451,-42.021
C02374=1018.914,74.097,-127.720,-24.288,21.451,-42.023
C02375=1018.916,73.886,-127.700,-24.287,21.452,-42.025
C02376=1018.919,73.465,-127.661,-24.287,21.452,-42.028
C02377=1018.923,73.048,-127.623,-24.286,21.452,-42.034
C02378=1018.926,72.632,-127.584,-24.285,21.452,-42.037
C02379=1018.930,72.219,-127.547,-24.285,21.453,-42.041
C02380=1018.933,71.807,-127.509,-24.285,21.453,-42.045
C02381=1018.937,71.396,-127.471,-24.284,21.454,-42.049
C02382=1018.940,70.984,-127.433,-24.283,21.453,-42.054
C02383=1018.944,70.573,-127.396,-24.283,21.454,-42.058
C02384=1018.946,70.162,-127.359,-24.282,21.454,-42.061
C02385=1018.950,69.751,-127.321,-24.282,21.455,-42.065
C02386=1018.953,69.341,-127.283,-24.281,21.455,-42.069
C02387=1018.956,68.932,-127.246,-24.280,21.455,-42.074
C02388=1018.960,68.525,-127.209,-24.280,21.456,-42.078
C02389=1018.963,68.119,-127.171,-24.279,21.456,-42.082
C02390=1018.967,67.714,-127.135,-24.279,21.457,-42.085
C02391=1018.970,67.311,-127.097,-24.278,21.457,-42.089
C02392=1018.973,66.909,-127.060,-24.278,21.457,-42.094
C02393=1018.975,66.507,-127.025,-24.277,21.457,-42.098
C02394=1018.979,66.110,-126.987,-24.277,21.458,-42.102
C02395=1018.982,65.701,-126.951,-24.276,21.458,-42.106
C02396=1018.983,65.488,-126.931,-24.276,21.459,-42.108
C02397=1018.985,65.268,-126.911,-24.275,21.458,-42.111
C02398=1018.987,65.037,-126.890,-24.275,21.458,-42.113
C02399=1018.989,64.802,-126.869,-24.275,21.459,-42.115
C02400=1018.991,64.566,-126.847,-24.274,21.459,-42.116
C02401=1018.992,64.336,-126.826,-24.274,21.459,-42.120
C02402=1018.994,64.118,-126.807,-24.274,21.460,-42.122
C02403=1018.996,63.911,-126.787,-24.274,21.460,-42.124
C02404=1018.997,63.695,-126.768,-24.273,21.459,-42.127
C02405=1018.999,63.444,-126.745,-24.273,21.460,-42.129
C02406=1019.001,63.177,-126.721,-24.272,21.460,-42.131
C02407=1019.003,62.924,-126.697,-24.272,21.460,-42.133
C02408=1019.006,62.504,-126.659,-24.271,21.461,-42.139
C02409=1019.009,62.104,-126.623,-24.271,21.461,-42.142
C02410=1019.012,61.704,-126.587,-24.270,21.462,-42.146
C02411=1019.015,61.304,-126.550,-24.270,21.462,-42.150
C02412=1019.018,60.903,-126.513,-24.269,21.462,-42.155
C02413=1019.021,60.503,-126.477,-24.269,21.463,-42.159
C02414=1019.023,60.103,-126.441,-24.268,21.463,-42.163
C02415=1019.027,59.703,-126.405,-24.268,21.464,-42.166
C02416=1019.029,59.302,-126.368,-24.267,21.463,-42.172
C02417=1019.032,58.902,-126.332,-24.266,21.464,-42.175
C02418=1019.035,58.502,-126.296,-24.266,21.464,-42.179
C02419=1019.038,58.102,-126.259,-24.265,21.465,-42.183
C02420=1019.041,57.702,-126.223,-24.264,21.465,-42.188
C02421=1019.043,57.301,-126.188,-24.264,21.465,-42.192
C02422=1019.046,56.901,-126.151,-24.264,21.466,-42.196
C02423=1019.049,56.500,-126.115,-24.263,21.465,-42.201
C02424=1019.052,56.101,-126.079,-24.262,21.467,-42.205
C02425=1019.054,55.700,-126.042,-24.262,21.467,-42.209
C02426=1019.058,55.300,-126.006,-24.261,21.468,-42.212
C02427=1019.059,54.900,-125.970,-24.260,21.468,-42.218
C02428=1019.062,54.500,-125.934,-24.260,21.468,-42.221
C02429=1019.065,54.100,-125.898,-24.259,21.468,-42.225
C02430=1019.068,53.700,-125.862,-24.259,21.468,-42.230
C02431=1019.070,53.299,-125.825,-24.258,21.469,-42.234
C02432=1019.073,52.900,-125.790,-24.258,21.469,-42.238
C02433=1019.075,52.498,-125.754,-24.257,21.469,-42.243
C02434=1019.079,52.099,-125.718,-24.256,21.470,-42.247
C02435=1019.080,51.698,-125.682,-24.256,21.471,-42.251
C02436=1019.083,51.299,-125.646,-24.255,21.471,-42.255
C02437=1019.086,50.898,-125.609,-24.255,21.471,-42.260
C02438=1019.088,50.498,-125.574,-24.254,21.472,-42.264
C02439=1019.091,50.098,-125.537,-24.254,21.472,-42.268
C02440=1019.093,49.698,-125.502,-24.253,21.472,-42.273
C02441=1019.096,49.297,-125.466,-24.252,21.473,-42.277
C02442=1019.099,48.897,-125.430,-24.251,21.472,-42.282
C02443=1019.100,48.497,-125.394,-24.251,21.474,-42.286
C02444=1019.104,48.097,-125.358,-24.251,21.474,-42.290
C02445=1019.105,47.697,-125.322,-24.250,21.474,-42.295
C02446=1019.108,47.297,-125.286,-24.249,21.475,-42.299
C02447=1019.110,46.897,-125.250,-24.249,21.475,-42.302
C02448=1019.113,46.497,-125.215,-24.248,21.475,-42.308
C02449=1019.115,46.096,-125.179,-24.247,21.475,-42.311
C02450=1019.117,45.697,-125.143,-24.247,21.477,-42.316
C02451=1019.120,45.297,-125.108,-24.246,21.477,-42.321
C02452=1019.122,44.897,-125.071,-24.246,21.477,-42.325
C02453=1019.125,44.497,-125.036,-24.245,21.477,-42.330
C02454=1019.127,44.096,-125.000,-24.244,21.477,-42.333
C02455=1019.129,43.697,-124.965,-24.244,21.479,-42.338
C02456=1019.131,43.296,-124.929,-24.243,21.479,-42.343
C02457=1019.134,42.897,-124.893,-24.243,21.479,-42.347
C02458=1019.135,42.496,-124.857,-24.242,21.479,-42.352
C02459=1019.138,42.097,-124.821,-24.241,21.479,-42.356
C02460=1019.140,41.696,-124.786,-24.241,21.480,-42.359
C02461=1019.142,41.296,-124.751,-24.240,21.481,-42.365
C02462=1019.144,40.897,-124.715,-24.240,21.481,-42.369
C02463=1019.146,40.497,-124.679,-24.239,21.481,-42.374
C02464=1019.149,40.097,-124.644,-24.238,21.481,-42.378
C02465=1019.151,39.696,-124.609,-24.238,21.482,-42.383
C02466=1019.153,39.297,-124.573,-24.237,21.483,-42.387
C02467=1019.155,38.897,-124.538,-24.237,21.483,-42.391
C02468=1019.157,38.497,-124.502,-24.236,21.483,-42.396
C02469=1019.159,38.097,-124.466,-24.235,21.483,-42.400
C02470=1019.161,37.697,-124.430,-24.235,21.484,-42.405
C02471=1019.164,37.297,-124.395,-24.234,21.485,-42.409
C02472=1019.165,36.898,-124.360,-24.233,21.484,-42.414
C02473=1019.167,36.497,-124.325,-24.233,21.485,-42.418
C02474=1019.169,36.098,-124.289,-24.232,21.486,-42.424
C02475=1019.172,35.698,-124.254,-24.231,21.486,-42.428
C02476=1019.173,35.298,-124.218,-24.231,21.486,-42.433
C02477=1019.175,34.898,-124.183,-24.230,21.486,-42.437
C02478=1019.178,34.499,-124.148,-24.229,21.487,-42.442
C02479=1019.179,34.099,-124.113,-24.229,21.488,-42.446
C02480=1019.181,33.699,-124.077,-24.228,21.487,-42.451
C02481=1019.182,33.300,-124.042,-24.228,21.489,-42.455
C02482=1019.184,32.900,-124.006,-24.227,21.489,-42.461
C02483=1019.186,32.501,-123.971,-24.226,21.489,-42.464
C02484=1019.188,32.100,-123.936,-24.226,21.489,-42.469
C02485=1019.190,31.701,-123.902,-24.225,21.490,-42.474
C02486=1019.192,31.301,-123.866,-24.224,21.490,-42.479
C02487=1019.193,30.902,-123.831,-24.224,21.491,-42.483
C02488=1019.195,30.503,-123.796,-24.223,21.491,-42.488
C02489=1019.197,30.103,-123.760,-24.223,21.492,-42.492
C02490=1019.199,29.704,-123.725,-24.222,21.492,-42.497
C02491=1019.200,29.303,-123.691,-24.221,21.492,-42.501
C02492=1019.202,28.904,-123.655,-24.221,21.493,-42.507
C02493=1019.204,28.505,-123.620,-24.220,21.493,-42.510
C02494=1019.206,28.105,-123.585,-24.219,21.493,-42.516
C02495=1019.207,27.706,-123.550,-24.219,21.495,-42.520
C02496=1019.209,27.307,-123.516,-24.218,21.494,-42.525
C02497=1019.210,26.908,-123.481,-24.218,21.495,-42.529
C02498=1019.212,26.507,-123.445,-24.217,21.496,-42.534
C02499=1019.214,26.108,-123.410,-24.216,21.496,-42.540
C02500=1019.215,25.709,-123.375,-24.215,21.496,-42.543
C02501=1019.217,25.309,-123.341,-24.215,21.497,-42.549
C02502=1019.219,24.910,-123.306,-24.214,21.497,-42.553
C02503=1019.220,24.511,-123.271,-24.213,21.497,-42.558
C02504=1019.221,24.128,-123.238,-24.213,21.498,-42.562
C02505=1019.223,23.797,-123.209,-24.213,21.498,-42.564
C02506=1019.223,23.527,-123.185,-24.212,21.498,-42.567
C02507=1019.224,23.292,-123.165,-24.211,21.499,-42.573
C02508=1019.225,23.060,-123.145,-24.211,21.500,-42.577
C02509=1019.227,22.794,-123.121,-24.211,21.500,-42.580
C02510=1019.228,22.471,-123.093,-24.210,21.500,-42.584
C02511=1019.229,22.097,-123.060,-24.210,21.501,-42.586
C02512=1019.230,21.683,-123.024,-24.209,21.501,-42.593
C02513=1019.231,21.439,-123.004,-24.208,21.501,-42.597
C02514=1019.232,21.166,-122.980,-24.208,21.502,-42.599
C02515=1019.233,20.875,-122.954,-24.207,21.501,-42.602
C02516=1019.235,20.578,-122.928,-24.207,21.501,-42.604
C02517=1019.236,20.291,-122.904,-24.207,21.503,-42.606
C02518=1019.236,20.026,-122.880,-24.206,21.502,-42.610
C02519=1019.237,19.788,-122.859,-24.206,21.503,-42.613
C02520=1019.237,19.578,-122.842,-24.205,21.503,-42.617
C02521=1019.238,19.180,-122.808,-24.205,21.503,-42.622
C02522=1019.240,18.785,-122.773,-24.204,21.503,-42.626
C02523=1019.241,18.389,-122.738,-24.203,21.504,-42.632
C02524=1019.242,17.994,-122.704,-24.203,21.505,-42.635
C02525=1019.244,17.599,-122.671,-24.202,21.505,-42.641
C02526=1019.245,17.206,-122.636,-24.201,21.505,-42.646
C02527=1019.246,16.813,-122.603,-24.201,21.506,-42.650
C02528=1019.247,16.421,-122.569,-24.200,21.506,-42.656
C02529=1019.249,16.030,-122.535,-24.200,21.507,-42.659
C02530=1019.250,15.640,-122.501,-24.199,21.507,-42.665
C02531=1019.251,15.251,-122.467,-24.198,21.508,-42.670
C02532=1019.253,14.862,-122.434,-24.198,21.508,-42.674
C02533=1019.253,14.474,-122.401,-24.197,21.509,-42.680
C02534=1019.255,14.085,-122.367,-24.196,21.509,-42.683
C02535=1019.255,13.699,-122.334,-24.196,21.509,-42.689
C02536=1019.257,13.312,-122.300,-24.195,21.511,-42.693
C02537=1019.258,12.925,-122.267,-24.194,21.510,-42.698
C02538=1019.259,12.539,-122.234,-24.193,21.510,-42.703
C02539=1019.260,12.152,-122.200,-24.193,21.512,-42.707
C02540=1019.261,11.766,-122.168,-24.192,21.511,-42.713
C02541=1019.263,11.380,-122.134,-24.192,21.512,-42.716
C02542=1019.263,10.997,-122.101,-24.191,21.513,-42.722
C02543=1019.264,10.616,-122.069,-24.191,21.513,-42.726
C02544=1019.265,10.237,-122.036,-24.190,21.513,-42.731
C02545=1019.265,9.861,-122.004,-24.189,21.514,-42.737
C02546=1019.267,9.485,-121.972,-24.189,21.514,-42.740
C02547=1019.267,9.110,-121.940,-24.188,21.515,-42.746
C02548=1019.269,8.731,-121.907,-24.187,21.515,-42.751
C02549=1019.270,8.351,-121.875,-24.187,21.516,-42.755
C02550=1019.270,7.967,-121.842,-24.186,21.516,-42.761
C02551=1019.271,7.579,-121.809,-24.185,21.517,-42.764
C02552=1019.272,7.188,-121.776,-24.185,21.517,-42.770
C02553=1019.272,6.796,-121.742,-24.184,21.517,-42.775
C02554=1019.274,6.403,-121.709,-24.183,21.519,-42.779
C02555=1019.274,6.010,-121.675,-24.182,21.518,-42.785
C02556=1019.275,5.615,-121.641,-24.182,21.519,-42.790
C02557=1019.276,5.220,-121.608,-24.181,21.520,-42.794
C02558=1019.276,4.825,-121.574,-24.180,21.519,-42.799
C02559=1019.277,4.428,-121.541,-24.180,21.520,-42.805
C02560=1019.278,4.039,-121.508,-24.179,21.521,-42.809
C02561=1019.279,3.680,-121.477,-24.179,21.521,-42.812
C02562=1019.280,3.352,-121.449,-24.178,21.521,-42.817
C02563=1019.280,3.039,-121.422,-24.177,21.522,-42.823
C02564=1019.281,2.716,-121.395,-24.177,21.522,-42.827
C02565=1019.281,2.363,-121.366,-24.176,21.523,-42.833
C02566=1019.282,1.977,-121.333,-24.175,21.524,-42.836
C02567=1019.282,1.580,-121.299,-24.175,21.523,-42.841
C02568=1019.283,1.180,-121.265,-24.174,21.525,-42.846
C02569=1019.283,0.780,-121.232,-24.173,21.525,-42.851
C02570=1019.284,0.379,-121.198,-24.173,21.525,-42.857
C02571=1019.285,-0.025,-121.164,-24.172,21.525,-42.862
C02572=1019.286,-0.430,-121.129,-24.171,21.526,-42.867
C02573=1019.285,-0.838,-121.095,-24.171,21.527,-42.872
C02574=1019.286,-1.248,-121.060,-24.170,21.527,-42.877
C02575=1019.287,-1.660,-121.025,-24.169,21.528,-42.882
C02576=1019.287,-2.076,-120.991,-24.169,21.529,-42.888
C02577=1019.287,-2.493,-120.955,-24.168,21.529,-42.893
C02578=1019.288,-2.912,-120.920,-24.167,21.529,-42.899
C02579=1019.289,-3.334,-120.885,-24.166,21.530,-42.904
C02580=1019.289,-3.545,-120.867,-24.166,21.530,-42.908
C02581=1019.289,-3.757,-120.849,-24.165,21.530,-42.910
C02582=1019.289,-3.970,-120.831,-24.165,21.530,-42.913
C02583=1019.290,-4.186,-120.813,-24.165,21.531,-42.915
C02584=1019.290,-4.403,-120.794,-24.164,21.531,-42.919
C02585=1019.290,-4.622,-120.776,-24.164,21.531,-42.921
C02586=1019.290,-4.842,-120.758,-24.163,21.532,-42.925
C02587=1019.290,-5.062,-120.739,-24.163,21.532,-42.927
C02588=1019.291,-5.285,-120.721,-24.163,21.532,-42.930
C02589=1019.291,-5.508,-120.701,-24.162,21.532,-42.934
C02590=1019.292,-5.733,-120.683,-24.162,21.533,-42.935
C02591=1019.291,-5.957,-120.664,-24.161,21.533,-42.939
C02592=1019.291,-6.181,-120.645,-24.161,21.533,-42.941
C02593=1019.292,-6.405,-120.627,-24.161,21.533,-42.944
C02594=1019.292,-6.628,-120.608,-24.160,21.534,-42.947
C02595=1019.292,-6.851,-120.590,-24.160,21.534,-42.950
C02596=1019.292,-7.072,-120.571,-24.160,21.535,-42.952
C02597=1019.292,-7.293,-120.552,-24.159,21.534,-42.956
C02598=1019.293,-7.512,-120.534,-24.159,21.535,-42.959
C02599=1019.293,-7.730,-120.516,-24.158,21.535,-42.961
C02600=1019.292,-7.947,-120.498,-24.158,21.536,-42.965
C02601=1019.293,-8.164,-120.479,-24.158,21.536,-42.967
C02602=1019.293,-8.380,-120.461,-24.157,21.536,-42.971
C02603=1019.293,-8.597,-120.443,-24.157,21.537,-42.973
C02604=1019.293,-8.814,-120.425,-24.156,21.536,-42.976
C02605=1019.294,-9.030,-120.407,-24.156,21.537,-42.980
C02606=1019.293,-9.247,-120.389,-24.156,21.537,-42.982
C02607=1019.294,-9.463,-120.371,-24.155,21.538,-42.985
C02608=1019.294,-9.680,-120.353,-24.155,21.538,-42.987
C02609=1019.294,-9.896,-120.335,-24.154,21.538,-42.991
C02610=1019.293,-10.111,-120.318,-24.154,21.539,-42.993
C02611=1019.293,-10.326,-120.299,-24.154,21.538,-42.996
C02612=1019.294,-10.541,-120.281,-24.153,21.539,-42.998
C02613=1019.294,-10.755,-120.264,-24.153,21.539,-43.002
C02614=1019.294,-10.969,-120.246,-24.152,21.539,-43.006
C02615=1019.294,-11.183,-120.228,-24.152,21.540,-43.007
C02616=1019.295,-11.397,-120.210,-24.152,21.540,-43.011
C02617=1019.294,-11.610,-120.193,-24.151,21.540,-43.013
C02618=1019.294,-11.822,-120.175,-24.151,21.540,-43.016
C02619=1019.294,-12.034,-120.158,-24.151,21.541,-43.019
C02620=1019.294,-12.245,-120.140,-24.150,21.541,-43.022
C02621=1019.294,-12.455,-120.122,-24.150,21.542,-43.024
C02622=1019.294,-12.876,-120.087,-24.149,21.542,-43.029
C02623=1019.294,-13.293,-120.053,-24.148,21.543,-43.035
C02624=1019.294,-13.708,-120.019,-24.148,21.543,-43.041
C02625=1019.294,-14.119,-119.984,-24.147,21.544,-43.046
C02626=1019.294,-14.528,-119.950,-24.146,21.544,-43.052
C02627=1019.294,-14.934,-119.917,-24.145,21.545,-43.057
C02628=1019.294,-15.337,-119.884,-24.145,21.545,-43.063
C02629=1019.294,-15.737,-119.851,-24.144,21.546,-43.068
C02630=1019.294,-16.137,-119.818,-24.143,21.546,-43.074
C02631=1019.294,-16.535,-119.785,-24.142,21.547,-43.079
C02632=1019.294,-16.933,-119.752,-24.142,21.548,-43.085
C02633=1019.294,-17.331,-119.720,-24.141,21.547,-43.090
C02634=1019.293,-17.741,-119.686,-24.140,21.548,-43.098
C02635=1019.293,-17.990,-119.665,-24.139,21.549,-43.101
C02636=1019.294,-18.277,-119.642,-24.139,21.549,-43.105
C02637=1019.293,-18.589,-119.616,-24.139,21.550,-43.107
C02638=1019.293,-18.901,-119.590,-24.139,21.550,-43.109
C02639=1019.292,-19.188,-119.566,-24.138,21.550,-43.113
C02640=1019.292,-19.437,-119.546,-24.138,21.551,-43.116
C02641=1019.292,-19.849,-119.512,-24.136,21.551,-43.123
C02642=1019.292,-20.246,-119.479,-24.136,21.552,-43.129
C02643=1019.291,-20.644,-119.447,-24.135,21.553,-43.135
C02644=1019.291,-21.041,-119.414,-24.134,21.552,-43.140
C02645=1019.291,-21.439,-119.382,-24.134,21.553,-43.146
C02646=1019.291,-21.836,-119.350,-24.133,21.554,-43.151
C02647=1019.291,-22.233,-119.317,-24.132,21.554,-43.156
C02648=1019.290,-22.631,-119.285,-24.131,21.555,-43.162
C02649=1019.290,-23.028,-119.252,-24.131,21.555,-43.168
C02650=1019.289,-23.425,-119.220,-24.130,21.556,-43.173
C02651=1019.289,-23.823,-119.187,-24.129,21.556,-43.178
C02652=1019.289,-24.221,-119.155,-24.128,21.557,-43.184
C02653=1019.288,-24.619,-119.122,-24.128,21.558,-43.190
C02654=1019.287,-25.016,-119.090,-24.127,21.558,-43.195
C02655=1019.287,-25.414,-119.057,-24.126,21.558,-43.201
C02656=1019.286,-25.811,-119.025,-24.125,21.559,-43.206
C02657=1019.286,-26.208,-118.993,-24.125,21.560,-43.212
C02658=1019.286,-26.606,-118.960,-24.124,21.560,-43.217
C02659=1019.285,-27.003,-118.928,-24.123,21.561,-43.221
C02660=1019.284,-27.401,-118.896,-24.123,21.562,-43.227
C02661=1019.283,-27.798,-118.864,-24.122,21.562,-43.232
C02662=1019.283,-28.196,-118.832,-24.121,21.562,-43.238
C02663=1019.283,-28.593,-118.799,-24.120,21.563,-43.243
C02664=1019.282,-28.990,-118.767,-24.120,21.564,-43.249
C02665=1019.281,-29.388,-118.735,-24.119,21.565,-43.255
C02666=1019.281,-29.786,-118.703,-24.118,21.565,-43.260
C02667=1019.280,-30.183,-118.671,-24.117,21.565,-43.265
C02668=1019.279,-30.581,-118.639,-24.117,21.566,-43.271
C02669=1019.278,-30.978,-118.607,-24.116,21.567,-43.277
C02670=1019.277,-31.375,-118.574,-24.115,21.568,-43.282
C02671=1019.277,-31.773,-118.543,-24.114,21.567,-43.287
C02672=1019.276,-32.170,-118.511,-24.114,21.568,-43.293
C02673=1019.275,-32.568,-118.479,-24.113,21.569,-43.299
C02674=1019.274,-32.965,-118.446,-24.112,21.570,-43.304
C02675=1019.274,-33.363,-118.415,-24.111,21.570,-43.310
C02676=1019.272,-33.760,-118.383,-24.111,21.570,-43.315
C02677=1019.271,-34.157,-118.351,-24.110,21.571,-43.321
C02678=1019.271,-34.554,-118.319,-24.109,21.571,-43.328
C02679=1019.270,-34.952,-118.287,-24.108,21.572,-43.334
C02680=1019.269,-35.349,-118.256,-24.107,21.572,-43.339
C02681=1019.268,-35.746,-118.224,-24.107,21.573,-43.344
C02682=1019.267,-36.144,-118.191,-24.106,21.573,-43.350
C02683=1019.265,-36.542,-118.160,-24.105,21.574,-43.356
C02684=1019.265,-36.939,-118.128,-24.105,21.575,-43.361
C02685=1019.263,-37.336,-118.096,-24.104,21.575,-43.366
C02686=1019.263,-37.734,-118.065,-24.103,21.576,-43.372
C02687=1019.262,-38.131,-118.033,-24.102,21.576,-43.378
C02688=1019.260,-38.528,-118.001,-24.102,21.577,-43.383
C02689=1019.259,-38.925,-117.970,-24.101,21.578,-43.389
C02690=1019.258,-39.323,-117.938,-24.100,21.578,-43.394
C02691=1019.257,-39.720,-117.907,-24.099,21.579,-43.400
C02692=1019.256,-40.117,-117.874,-24.099,21.579,-43.405
C02693=1019.255,-40.514,-117.844,-24.098,21.580,-43.411
C02694=1019.253,-40.911,-117.812,-24.097,21.581,-43.417
C02695=1019.253,-41.308,-117.780,-24.096,21.582,-43.422
C02696=1019.251,-41.706,-117.749,-24.096,21.582,-43.427
C02697=1019.250,-42.103,-117.717,-24.095,21.582,-43.433
C02698=1019.249,-42.501,-117.686,-24.094,21.583,-43.439
C02699=1019.248,-42.898,-117.654,-24.093,21.584,-43.444
C02700=1019.246,-43.295,-117.623,-24.092,21.584,-43.451
C02701=1019.245,-43.692,-117.592,-24.092,21.585,-43.457
C02702=1019.244,-44.089,-117.560,-24.091,21.585,-43.462
C02703=1019.242,-44.486,-117.529,-24.090,21.585,-43.468
C02704=1019.240,-44.884,-117.497,-24.089,21.586,-43.473
C02705=1019.239,-45.281,-117.466,-24.089,21.587,-43.479
C02706=1019.237,-45.678,-117.434,-24.088,21.588,-43.485
C02707=1019.236,-46.076,-117.403,-24.087,21.589,-43.490
C02708=1019.235,-46.473,-117.372,-24.086,21.588,-43.496
C02709=1019.233,-46.870,-117.341,-24.086,21.589,-43.501
C02710=1019.231,-47.267,-117.310,-24.085,21.590,-43.507
C02711=1019.230,-47.664,-117.278,-24.084,21.591,-43.512
C02712=1019.229,-48.061,-117.247,-24.084,21.592,-43.518
C02713=1019.227,-48.458,-117.216,-24.083,21.592,-43.525
C02714=1019.226,-48.856,-117.185,-24.082,21.592,-43.531
C02715=1019.224,-49.252,-117.154,-24.081,21.592,-43.536
C02716=1019.222,-49.649,-117.122,-24.080,21.593,-43.542
C02717=1019.221,-50.046,-117.092,-24.080,21.594,-43.547
C02718=1019.219,-50.443,-117.061,-24.079,21.595,-43.553
C02719=1019.218,-50.840,-117.030,-24.078,21.595,-43.558
C02720=1019.216,-51.237,-116.999,-24.077,21.596,-43.564
C02721=1019.214,-51.634,-116.967,-24.077,21.597,-43.570
C02722=1019.212,-52.031,-116.937,-24.076,21.598,-43.575
C02723=1019.211,-52.428,-116.906,-24.075,21.598,-43.581
C02724=1019.209,-52.825,-116.875,-24.074,21.598,-43.588
C02725=1019.207,-53.222,-116.844,-24.073,21.599,-43.593
C02726=1019.205,-53.619,-116.813,-24.073,21.599,-43.599
C02727=1019.204,-54.015,-116.783,-24.072,21.600,-43.604
C02728=1019.202,-54.412,-116.752,-24.071,21.601,-43.610
C02729=1019.200,-54.809,-116.721,-24.071,21.602,-43.616
C02730=1019.198,-55.206,-116.690,-24.070,21.603,-43.621
C02731=1019.196,-55.604,-116.659,-24.069,21.602,-43.627
C02732=1019.194,-56.002,-116.628,-24.068,21.603,-43.632
C02733=1019.192,-56.400,-116.598,-24.067,21.603,-43.639
C02734=1019.191,-56.797,-116.567,-24.067,21.604,-43.645
C02735=1019.188,-57.195,-116.536,-24.066,21.605,-43.651
C02736=1019.186,-57.594,-116.505,-24.065,21.606,-43.656
C02737=1019.184,-57.993,-116.474,-24.064,21.606,-43.662
C02738=1019.182,-58.393,-116.443,-24.064,21.607,-43.667
C02739=1019.180,-58.793,-116.413,-24.063,21.608,-43.673
C02740=1019.178,-59.194,-116.381,-24.062,21.608,-43.680
C02741=1019.175,-59.595,-116.350,-24.061,21.609,-43.686
C02742=1019.173,-59.998,-116.319,-24.061,21.610,-43.691
C02743=1019.171,-60.400,-116.288,-24.060,21.610,-43.697
C02744=1019.169,-60.802,-116.257,-24.059,21.610,-43.702
C02745=1019.167,-61.206,-116.227,-24.058,21.611,-43.708
C02746=1019.165,-61.610,-116.196,-24.057,21.611,-43.715
C02747=1019.163,-62.015,-116.165,-24.057,21.612,-43.720
C02748=1019.160,-62.420,-116.134,-24.056,21.613,-43.726
C02749=1019.157,-62.825,-116.102,-24.055,21.614,-43.732
C02750=1019.155,-63.232,-116.071,-24.054,21.615,-43.737
C02751=1019.153,-63.639,-116.040,-24.053,21.615,-43.744
C02752=1019.150,-64.046,-116.009,-24.053,21.615,-43.750
C02753=1019.148,-64.454,-115.978,-24.052,21.616,-43.756
C02754=1019.146,-64.862,-115.947,-24.051,21.617,-43.761
C02755=1019.143,-65.270,-115.915,-24.050,21.617,-43.768
C02756=1019.140,-65.679,-115.885,-24.049,21.618,-43.774
C02757=1019.138,-66.088,-115.853,-24.049,21.619,-43.780
C02758=1019.136,-66.497,-115.822,-24.048,21.620,-43.785
C02759=1019.133,-66.907,-115.791,-24.047,21.620,-43.791
C02760=1019.130,-67.317,-115.760,-24.046,21.621,-43.798
C02761=1019.127,-67.727,-115.728,-24.046,21.621,-43.804
C02762=1019.125,-68.138,-115.697,-24.045,21.622,-43.809
C02763=1019.123,-68.548,-115.666,-24.044,21.623,-43.815
C02764=1019.120,-68.959,-115.635,-24.043,21.623,-43.822
C02765=1019.117,-69.370,-115.603,-24.042,21.624,-43.827
C02766=1019.114,-69.780,-115.573,-24.042,21.625,-43.833
C02767=1019.112,-70.192,-115.541,-24.041,21.625,-43.839
C02768=1019.109,-70.602,-115.511,-24.040,21.626,-43.846
C02769=1019.106,-71.013,-115.479,-24.039,21.626,-43.851
C02770=1019.103,-71.425,-115.448,-24.039,21.627,-43.857
C02771=1019.100,-71.835,-115.417,-24.038,21.628,-43.865
C02772=1019.097,-72.247,-115.386,-24.037,21.629,-43.870
C02773=1019.094,-72.657,-115.355,-24.036,21.630,-43.876
C02774=1019.091,-73.068,-115.324,-24.035,21.631,-43.881
C02775=1019.089,-73.479,-115.294,-24.034,21.631,-43.888
C02776=1019.086,-73.889,-115.262,-24.034,21.632,-43.894
C02777=1019.083,-74.300,-115.231,-24.033,21.632,-43.900
C02778=1019.079,-74.710,-115.201,-24.032,21.633,-43.905
C02779=1019.077,-75.120,-115.170,-24.031,21.633,-43.912
C02780=1019.074,-75.529,-115.140,-24.031,21.634,-43.918
C02781=1019.071,-75.939,-115.108,-24.030,21.635,-43.924
C02782=1019.067,-76.349,-115.078,-24.029,21.636,-43.929
C02783=1019.064,-76.758,-115.047,-24.028,21.636,-43.936
C02784=1019.061,-77.166,-115.016,-24.027,21.637,-43.942
C02785=1019.059,-77.574,-114.986,-24.027,21.637,-43.948
C02786=1019.055,-77.983,-114.956,-24.026,21.638,-43.953
C02787=1019.052,-78.390,-114.925,-24.025,21.638,-43.960
C02788=1019.048,-78.797,-114.894,-24.024,21.639,-43.966
C02789=1019.045,-79.203,-114.864,-24.023,21.640,-43.972
C02790=1019.042,-79.610,-114.834,-24.023,21.641,-43.977
C02791=1019.038,-80.015,-114.804,-24.022,21.641,-43.984
C02792=1019.035,-80.421,-114.774,-24.021,21.642,-43.990
C02793=1019.032,-80.825,-114.743,-24.020,21.643,-43.995
C02794=1019.029,-81.229,-114.714,-24.020,21.643,-44.001
C02795=1019.025,-81.632,-114.684,-24.019,21.644,-44.007
C02796=1019.022,-82.035,-114.654,-24.018,21.644,-44.014
C02797=1019.018,-82.437,-114.624,-24.017,21.645,-44.019
C02798=1019.015,-82.839,-114.594,-24.016,21.646,-44.025
C02799=1019.012,-83.239,-114.564,-24.016,21.647,-44.031
C02800=1019.008,-83.640,-114.535,-24.015,21.648,-44.036
C02801=1019.005,-84.040,-114.505,-24.014,21.648,-44.043
C02802=1019.001,-84.446,-114.475,-24.013,21.649,-44.049
C02803=1018.999,-84.669,-114.458,-24.013,21.649,-44.053
C02804=1018.997,-84.910,-114.441,-24.012,21.650,-44.056
C02805=1018.995,-85.164,-114.422,-24.012,21.649,-44.060
C02806=1018.993,-85.418,-114.403,-24.012,21.650,-44.062
C02807=1018.990,-85.665,-114.384,-24.011,21.650,-44.065
C02808=1018.988,-85.895,-114.368,-24.011,21.651,-44.069
C02809=1018.985,-86.304,-114.338,-24.010,21.652,-44.077
C02810=1018.981,-86.692,-114.309,-24.009,21.652,-44.082
C02811=1018.978,-87.071,-114.281,-24.008,21.652,-44.087
C02812=1018.974,-87.444,-114.254,-24.007,21.653,-44.093
C02813=1018.970,-87.815,-114.226,-24.007,21.654,-44.099
C02814=1018.967,-88.191,-114.198,-24.006,21.655,-44.104
C02815=1018.963,-88.598,-114.169,-24.005,21.656,-44.112
C02816=1018.961,-88.846,-114.151,-24.005,21.656,-44.116
C02817=1018.958,-89.119,-114.130,-24.004,21.657,-44.117
C02818=1018.956,-89.404,-114.109,-24.004,21.656,-44.121
C02819=1018.953,-89.680,-114.090,-24.003,21.657,-44.124
C02820=1018.950,-89.929,-114.071,-24.003,21.657,-44.128
C02821=1018.949,-90.148,-114.055,-24.002,21.658,-44.132
C02822=1018.945,-90.544,-114.026,-24.002,21.659,-44.138
C02823=1018.941,-90.937,-113.997,-24.001,21.659,-44.145
C02824=1018.938,-91.330,-113.969,-24.000,21.660,-44.150
C02825=1018.934,-91.722,-113.940,-23.999,21.660,-44.156
C02826=1018.930,-92.114,-113.911,-23.999,21.661,-44.162
C02827=1018.925,-92.505,-113.883,-23.998,21.662,-44.167
C02828=1018.922,-92.894,-113.854,-23.997,21.663,-44.173
C02829=1018.917,-93.283,-113.825,-23.996,21.664,-44.178
C02830=1018.914,-93.672,-113.797,-23.996,21.664,-44.184
C02831=1018.910,-94.059,-113.769,-23.995,21.664,-44.189
C02832=1018.906,-94.446,-113.741,-23.994,21.665,-44.195
C02833=1018.902,-94.833,-113.713,-23.994,21.666,-44.200
C02834=1018.898,-95.217,-113.685,-23.993,21.666,-44.207
C02835=1018.894,-95.603,-113.657,-23.992,21.667,-44.213
C02836=1018.890,-95.987,-113.629,-23.991,21.668,-44.219
C02837=1018.886,-96.371,-113.601,-23.990,21.668,-44.224
C02838=1018.882,-96.755,-113.573,-23.990,21.669,-44.230
C02839=1018.878,-97.138,-113.546,-23.989,21.669,-44.235
C02840=1018.874,-97.522,-113.518,-23.988,21.670,-44.241
C02841=1018.869,-97.904,-113.490,-23.988,21.671,-44.246
C02842=1018.865,-98.289,-113.462,-23.987,21.672,-44.252
C02843=1018.861,-98.671,-113.435,-23.986,21.673,-44.258
C02844=1018.857,-99.056,-113.407,-23.985,21.673,-44.263
C02845=1018.852,-99.439,-113.379,-23.985,21.673,-44.268
C02846=1018.848,-99.823,-113.351,-23.984,21.674,-44.274
C02847=1018.844,-100.207,-113.323,-23.983,21.675,-44.280
C02848=1018.840,-100.593,-113.296,-23.982,21.676,-44.285
C02849=1018.836,-100.978,-113.267,-23.982,21.677,-44.291
C02850=1018.831,-101.364,-113.240,-23.981,21.676,-44.296
C02851=1018.827,-101.752,-113.212,-23.980,21.677,-44.302
C02852=1018.822,-102.140,-113.184,-23.980,21.678,-44.307
C02853=1018.817,-102.528,-113.156,-23.979,21.678,-44.314
C02854=1018.813,-102.917,-113.128,-23.978,21.679,-44.320
C02855=1018.809,-103.306,-113.100,-23.977,21.680,-44.326
C02856=1018.804,-103.697,-113.073,-23.976,21.681,-44.331
C02857=1018.799,-104.089,-113.044,-23.976,21.682,-44.337
C02858=1018.795,-104.480,-113.016,-23.975,21.681,-44.342
C02859=1018.790,-104.871,-112.988,-23.974,21.682,-44.348
C02860=1018.785,-105.264,-112.960,-23.974,21.683,-44.353
C02861=1018.781,-105.656,-112.932,-23.973,21.684,-44.359
C02862=1018.776,-106.050,-112.904,-23.972,21.685,-44.365
C02863=1018.771,-106.443,-112.876,-23.971,21.686,-44.370
C02864=1018.766,-106.836,-112.848,-23.971,21.686,-44.376
C02865=1018.761,-107.229,-112.820,-23.970,21.687,-44.383
C02866=1018.757,-107.622,-112.791,-23.969,21.687,-44.388
C02867=1018.753,-108.014,-112.763,-23.968,21.688,-44.394
C02868=1018.747,-108.407,-112.735,-23.968,21.688,-44.399
C02869=1018.742,-108.800,-112.707,-23.967,21.689,-44.405
C02870=1018.737,-109.193,-112.679,-23.966,21.690,-44.411
C02871=1018.732,-109.586,-112.651,-23.965,21.691,-44.416
C02872=1018.727,-109.979,-112.623,-23.965,21.691,-44.422
C02873=1018.722,-110.372,-112.595,-23.964,21.692,-44.427
C02874=1018.717,-110.764,-112.567,-23.963,21.693,-44.433
C02875=1018.712,-111.156,-112.540,-23.963,21.694,-44.439
C02876=1018.707,-111.549,-112.512,-23.962,21.694,-44.446
C02877=1018.702,-111.942,-112.484,-23.961,21.694,-44.451
C02878=1018.697,-112.335,-112.456,-23.960,21.695,-44.456
C02879=1018.691,-112.727,-112.428,-23.959,21.696,-44.462
C02880=1018.686,-113.120,-112.400,-23.959,21.696,-44.468
C02881=1018.681,-113.513,-112.372,-23.958,21.697,-44.473
C02882=1018.676,-113.905,-112.345,-23.957,21.698,-44.479
C02883=1018.671,-114.298,-112.317,-23.957,21.699,-44.485
C02884=1018.665,-114.690,-112.289,-23.956,21.700,-44.490
C02885=1018.660,-115.082,-112.261,-23.955,21.701,-44.496
C02886=1018.654,-115.475,-112.234,-23.954,21.700,-44.501
C02887=1018.648,-115.867,-112.206,-23.954,21.701,-44.507
C02888=1018.644,-116.259,-112.178,-23.953,21.702,-44.512
C02889=1018.638,-116.652,-112.150,-23.952,21.703,-44.518
C02890=1018.632,-117.044,-112.123,-23.952,21.704,-44.523
C02891=1018.627,-117.436,-112.096,-23.951,21.705,-44.529
C02892=1018.622,-117.829,-112.067,-23.950,21.705,-44.536
C02893=1018.616,-118.221,-112.040,-23.949,21.705,-44.541
C02894=1018.611,-118.613,-112.013,-23.948,21.706,-44.547
C02895=1018.604,-119.005,-111.985,-23.948,21.706,-44.553
C02896=1018.599,-119.398,-111.957,-23.947,21.707,-44.558
C02897=1018.593,-119.790,-111.930,-23.946,21.708,-44.564
C02898=1018.587,-120.182,-111.902,-23.946,21.709,-44.569
C02899=1018.582,-120.574,-111.875,-23.945,21.710,-44.575
C02900=1018.576,-120.966,-111.847,-23.944,21.710,-44.580
C02901=1018.570,-121.358,-111.820,-23.943,21.710,-44.586
C02902=1018.565,-121.750,-111.793,-23.943,21.711,-44.591
C02903=1018.558,-122.142,-111.765,-23.942,21.712,-44.597
C02904=1018.552,-122.535,-111.738,-23.941,21.713,-44.603
C02905=1018.547,-122.926,-111.710,-23.941,21.714,-44.608
C02906=1018.541,-123.319,-111.682,-23.940,21.715,-44.614
C02907=1018.534,-123.711,-111.655,-23.939,21.714,-44.619
C02908=1018.529,-124.102,-111.628,-23.939,21.715,-44.625
C02909=1018.523,-124.495,-111.600,-23.938,21.716,-44.630
C02910=1018.517,-124.886,-111.573,-23.937,21.717,-44.636
C02911=1018.511,-125.279,-111.546,-23.936,21.718,-44.642
C02912=1018.506,-125.619,-111.523,-23.936,21.718,-44.647
C02913=1018.500,-125.959,-111.498,-23.935,21.719,-44.651
C02914=1018.499,-126.062,-111.491,-23.935,21.719,-44.652
C02915=1018.492,-126.454,-111.464,-23.934,21.719,-44.658
C02916=1018.486,-126.847,-111.437,-23.934,21.720,-44.664
C02917=1018.480,-127.238,-111.409,-23.933,21.721,-44.669
C02918=1018.474,-127.630,-111.382,-23.932,21.722,-44.675
C02919=1018.467,-128.022,-111.355,-23.932,21.723,-44.680
C02920=1018.462,-128.414,-111.328,-23.931,21.723,-44.686
C02921=1018.455,-128.806,-111.300,-23.930,21.723,-44.691
C02922=1018.448,-129.198,-111.274,-23.929,21.724,-44.697
C02923=1018.442,-129.589,-111.246,-23.929,21.725,-44.703
C02924=1018.435,-129.981,-111.219,-23.928,21.726,-44.708
C02925=1018.429,-130.373,-111.192,-23.927,21.727,-44.714
C02926=1018.423,-130.764,-111.165,-23.926,21.727,-44.719
C02927=1018.416,-131.156,-111.138,-23.926,21.728,-44.725
C02928=1018.409,-131.548,-111.111,-23.925,21.728,-44.730
C02929=1018.403,-131.940,-111.084,-23.924,21.729,-44.736
C02930=1018.396,-132.331,-111.057,-23.924,21.730,-44.741
C02931=1018.390,-132.723,-111.029,-23.923,21.730,-44.747
C02932=1018.383,-133.116,-111.002,-23.922,21.731,-44.752
C02933=1018.377,-133.507,-110.975,-23.922,21.732,-44.758
C02934=1018.370,-133.899,-110.948,-23.921,21.732,-44.763
C02935=1018.750,-133.871,-111.185,-23.921,21.732,-44.763
C02936=1018.757,-133.479,-111.212,-23.922,21.732,-44.758
C02937=1018.763,-133.088,-111.239,-23.922,21.731,-44.752
C02938=1018.769,-132.696,-111.266,-23.923,21.730,-44.747
C02939=1018.776,-132.304,-111.294,-23.924,21.730,-44.741
C02940=1018.782,-131.912,-111.320,-23.924,21.729,-44.736
C02941=1018.789,-131.521,-111.347,-23.925,21.728,-44.730
C02942=1018.795,-131.129,-111.374,-23.926,21.728,-44.725
C02943=1018.802,-130.737,-111.401,-23.926,21.727,-44.719
C02944=1018.808,-130.346,-111.428,-23.927,21.727,-44.714
C02945=1018.814,-129.954,-111.455,-23.928,21.726,-44.708
C02946=1018.821,-129.562,-111.482,-23.929,21.725,-44.703
C02947=1018.827,-129.170,-111.509,-23.929,21.724,-44.697
C02948=1018.834,-128.778,-111.536,-23.930,21.723,-44.691
C02949=1018.839,-128.386,-111.563,-23.931,21.723,-44.686
C02950=1018.846,-127.994,-111.591,-23.932,21.723,-44.680
C02951=1018.852,-127.603,-111.617,-23.932,21.722,-44.675
C02952=1018.858,-127.211,-111.645,-23.933,21.721,-44.669
C02953=1018.864,-126.819,-111.672,-23.934,21.720,-44.664
C02954=1018.870,-126.427,-111.700,-23.934,21.719,-44.658
C02955=1018.876,-126.035,-111.727,-23.935,21.719,-44.652
C02956=1018.882,-125.643,-111.754,-23.936,21.719,-44.647
C02957=1018.888,-125.251,-111.781,-23.936,21.718,-44.642
C02958=1018.894,-124.859,-111.808,-23.937,21.717,-44.636
C02959=1018.900,-124.467,-111.836,-23.938,21.716,-44.630
C02960=1018.906,-124.075,-111.863,-23.939,21.715,-44.625
C02961=1018.911,-123.683,-111.890,-23.939,21.714,-44.619
C02962=1018.918,-123.292,-111.917,-23.940,21.715,-44.614
C02963=1018.924,-122.899,-111.945,-23.941,21.714,-44.608
C02964=1018.929,-122.507,-111.972,-23.941,21.713,-44.603
C02965=1018.935,-122.115,-112.000,-23.942,21.712,-44.597
C02966=1018.941,-121.724,-112.026,-23.943,21.711,-44.591
C02967=1018.947,-121.331,-112.054,-23.943,21.710,-44.586
C02968=1018.952,-120.940,-112.082,-23.944,21.710,-44.580
C02969=1018.958,-120.547,-112.109,-23.945,21.710,-44.575
C02970=1018.964,-120.154,-112.136,-23.946,21.709,-44.569
C02971=1018.969,-119.763,-112.164,-23.946,21.708,-44.564
C02972=1018.975,-119.370,-112.192,-23.947,21.707,-44.558
C02973=1018.980,-118.978,-112.219,-23.948,21.706,-44.553
C02974=1018.986,-118.586,-112.246,-23.948,21.706,-44.547
C02975=1018.991,-118.194,-112.274,-23.949,21.705,-44.541
C02976=1018.996,-117.801,-112.302,-23.950,21.705,-44.536
C02977=1019.002,-117.409,-112.329,-23.951,21.705,-44.529
C02978=1019.007,-117.017,-112.356,-23.952,21.704,-44.523
C02979=1019.014,-116.625,-112.384,-23.952,21.703,-44.518
C02980=1019.018,-116.232,-112.412,-23.953,21.702,-44.512
C02981=1019.024,-115.840,-112.439,-23.954,21.701,-44.507
C02982=1019.028,-115.447,-112.467,-23.954,21.700,-44.501
C02983=1019.034,-115.055,-112.494,-23.955,21.701,-44.496
C02984=1019.039,-114.662,-112.523,-23.956,21.700,-44.490
C02985=1019.045,-114.270,-112.550,-23.957,21.699,-44.485
C02986=1019.050,-113.877,-112.578,-23.957,21.698,-44.479
C02987=1019.055,-113.486,-112.605,-23.958,21.697,-44.473
C02988=1019.060,-113.093,-112.633,-23.959,21.696,-44.468
C02989=1019.066,-112.700,-112.661,-23.959,21.696,-44.462
C02990=1019.070,-112.308,-112.688,-23.960,21.695,-44.456
C02991=1019.076,-111.915,-112.717,-23.961,21.694,-44.451
C02992=1019.081,-111.522,-112.745,-23.962,21.694,-44.446
C02993=1019.085,-111.130,-112.773,-23.963,21.694,-44.439
C02994=1019.091,-110.737,-112.800,-23.963,21.693,-44.433
C02995=1019.096,-110.344,-112.828,-23.964,21.692,-44.427
C02996=1019.101,-109.951,-112.856,-23.965,21.691,-44.422
C02997=1019.105,-109.559,-112.884,-23.965,21.691,-44.416
C02998=1019.110,-109.166,-112.912,-23.966,21.690,-44.411
C02999=1019.115,-108.773,-112.940,-23.967,21.689,-44.405
C03000=1019.121,-108.380,-112.968,-23.968,21.688,-44.399
C03001=1019.125,-107.988,-112.995,-23.968,21.688,-44.394
C03002=1019.129,-107.595,-113.024,-23.969,21.687,-44.388
C03003=1019.134,-107.202,-113.052,-23.970,21.687,-44.383
C03004=1019.139,-106.809,-113.080,-23.971,21.686,-44.376
C03005=1019.144,-106.416,-113.108,-23.971,21.686,-44.370
C03006=1019.148,-106.023,-113.136,-23.972,21.685,-44.365
C03007=1019.153,-105.630,-113.164,-23.973,21.684,-44.359
C03008=1019.158,-105.237,-113.192,-23.974,21.683,-44.353
C03009=1019.163,-104.845,-113.220,-23.974,21.682,-44.348
C03010=1019.168,-104.453,-113.248,-23.975,21.681,-44.342
C03011=1019.172,-104.061,-113.276,-23.976,21.682,-44.337
C03012=1019.176,-103.670,-113.304,-23.976,21.681,-44.331
C03013=1019.181,-103.280,-113.332,-23.977,21.680,-44.326
C03014=1019.185,-102.890,-113.360,-23.978,21.679,-44.320
C03015=1019.190,-102.501,-113.388,-23.979,21.678,-44.314
C03016=1019.194,-102.113,-113.415,-23.980,21.678,-44.307
C03017=1019.198,-101.725,-113.443,-23.980,21.677,-44.302
C03018=1019.203,-101.337,-113.472,-23.981,21.676,-44.296
C03019=1019.207,-100.952,-113.500,-23.982,21.677,-44.291
C03020=1019.212,-100.566,-113.528,-23.982,21.676,-44.285
C03021=1019.215,-100.181,-113.555,-23.983,21.675,-44.280
C03022=1019.220,-99.796,-113.583,-23.984,21.674,-44.274
C03023=1019.224,-99.412,-113.610,-23.985,21.673,-44.268
C03024=1019.228,-99.028,-113.638,-23.985,21.673,-44.263
C03025=1019.233,-98.645,-113.665,-23.986,21.673,-44.258
C03026=1019.237,-98.261,-113.694,-23.987,21.672,-44.252
C03027=1019.241,-97.878,-113.721,-23.988,21.671,-44.246
C03028=1019.244,-97.495,-113.749,-23.988,21.670,-44.241
C03029=1019.249,-97.111,-113.776,-23.989,21.669,-44.235
C03030=1019.253,-96.729,-113.804,-23.990,21.669,-44.230
C03031=1019.256,-96.344,-113.832,-23.990,21.668,-44.224
C03032=1019.260,-95.960,-113.860,-23.991,21.668,-44.219
C03033=1019.264,-95.576,-113.888,-23.992,21.667,-44.213
C03034=1019.269,-95.191,-113.916,-23.993,21.666,-44.207
C03035=1019.273,-94.805,-113.944,-23.994,21.666,-44.200
C03036=1019.276,-94.419,-113.972,-23.994,21.665,-44.195
C03037=1019.280,-94.033,-114.000,-23.995,21.664,-44.189
C03038=1019.285,-93.645,-114.028,-23.996,21.664,-44.184
C03039=1019.288,-93.257,-114.057,-23.996,21.664,-44.178
C03040=1019.292,-92.867,-114.085,-23.997,21.663,-44.173
C03041=1019.296,-92.477,-114.113,-23.998,21.662,-44.167
C03042=1019.299,-92.086,-114.142,-23.999,21.661,-44.162
C03043=1019.304,-91.695,-114.170,-23.999,21.660,-44.156
C03044=1019.308,-91.303,-114.199,-24.000,21.660,-44.150
C03045=1019.311,-90.910,-114.228,-24.001,21.659,-44.145
C03046=1019.315,-90.517,-114.256,-24.002,21.659,-44.138
C03047=1019.318,-90.121,-114.285,-24.002,21.658,-44.132
C03048=1019.321,-89.902,-114.302,-24.003,21.657,-44.128
C03049=1019.323,-89.652,-114.320,-24.003,21.657,-44.124
C03050=1019.325,-89.378,-114.340,-24.004,21.656,-44.121
C03051=1019.328,-89.093,-114.361,-24.004,21.657,-44.117
C03052=1019.330,-88.818,-114.381,-24.005,21.656,-44.116
C03053=1019.333,-88.572,-114.399,-24.005,21.656,-44.112
C03054=1019.336,-88.164,-114.429,-24.006,21.655,-44.104
C03055=1019.340,-87.788,-114.457,-24.007,21.654,-44.099
C03056=1019.343,-87.417,-114.484,-24.007,21.653,-44.093
C03057=1019.348,-87.044,-114.511,-24.008,21.652,-44.087
C03058=1019.351,-86.665,-114.539,-24.009,21.652,-44.082
C03059=1019.354,-86.277,-114.568,-24.010,21.652,-44.077
C03060=1019.357,-85.868,-114.598,-24.011,21.651,-44.069
C03061=1019.360,-85.638,-114.615,-24.011,21.650,-44.065
C03062=1019.361,-85.392,-114.633,-24.012,21.650,-44.062
C03063=1019.364,-85.137,-114.652,-24.012,21.649,-44.060
C03064=1019.366,-84.884,-114.670,-24.012,21.650,-44.056
C03065=1019.369,-84.642,-114.688,-24.013,21.649,-44.053
C03066=1019.371,-84.419,-114.705,-24.013,21.649,-44.049
C03067=1019.373,-84.013,-114.735,-24.014,21.648,-44.043
C03068=1019.378,-83.613,-114.765,-24.015,21.648,-44.036
C03069=1019.380,-83.213,-114.795,-24.016,21.647,-44.031
C03070=1019.384,-82.812,-114.824,-24.016,21.646,-44.025
C03071=1019.387,-82.411,-114.853,-24.017,21.645,-44.019
C03072=1019.391,-82.008,-114.884,-24.018,21.644,-44.014
C03073=1019.394,-81.605,-114.913,-24.019,21.644,-44.007
C03074=1019.397,-81.202,-114.943,-24.020,21.643,-44.001
C03075=1019.401,-80.798,-114.974,-24.020,21.643,-43.995
C03076=1019.404,-80.394,-115.004,-24.021,21.642,-43.990
C03077=1019.407,-79.989,-115.033,-24.022,21.641,-43.984
C03078=1019.410,-79.583,-115.064,-24.023,21.641,-43.977
C03079=1019.414,-79.177,-115.094,-24.023,21.640,-43.972
C03080=1019.417,-78.770,-115.124,-24.024,21.639,-43.966
C03081=1019.420,-78.363,-115.155,-24.025,21.638,-43.960
C03082=1019.423,-77.956,-115.186,-24.026,21.638,-43.953
C03083=1019.426,-77.548,-115.215,-24.027,21.637,-43.948
C03084=1019.429,-77.139,-115.246,-24.027,21.637,-43.942
C03085=1019.432,-76.731,-115.276,-24.028,21.636,-43.936
C03086=1019.436,-76.322,-115.308,-24.029,21.636,-43.929
C03087=1019.439,-75.912,-115.338,-24.030,21.635,-43.924
C03088=1019.441,-75.503,-115.369,-24.031,21.634,-43.918
C03089=1019.445,-75.093,-115.399,-24.031,21.633,-43.912
C03090=1019.447,-74.683,-115.431,-24.032,21.633,-43.905
C03091=1019.451,-74.273,-115.461,-24.033,21.632,-43.900
C03092=1019.453,-73.862,-115.492,-24.034,21.632,-43.894
C03093=1019.456,-73.452,-115.522,-24.034,21.631,-43.888
C03094=1019.459,-73.041,-115.554,-24.035,21.631,-43.881
C03095=1019.462,-72.631,-115.585,-24.036,21.630,-43.876
C03096=1019.465,-72.219,-115.616,-24.037,21.629,-43.870
C03097=1019.468,-71.809,-115.646,-24.038,21.628,-43.865
C03098=1019.471,-71.398,-115.678,-24.039,21.627,-43.857
C03099=1019.473,-70.987,-115.709,-24.039,21.626,-43.851
C03100=1019.477,-70.576,-115.740,-24.040,21.626,-43.846
C03101=1019.479,-70.165,-115.770,-24.041,21.625,-43.839
C03102=1019.481,-69.754,-115.802,-24.042,21.625,-43.833
C03103=1019.484,-69.343,-115.833,-24.042,21.624,-43.827
C03104=1019.487,-68.932,-115.864,-24.043,21.623,-43.822
C03105=1019.490,-68.522,-115.895,-24.044,21.623,-43.815
C03106=1019.492,-68.111,-115.927,-24.045,21.622,-43.809
C03107=1019.495,-67.701,-115.958,-24.046,21.621,-43.804
C03108=1019.497,-67.291,-115.988,-24.046,21.621,-43.798
C03109=1019.500,-66.881,-116.020,-24.047,21.620,-43.791
C03110=1019.502,-66.471,-116.051,-24.048,21.620,-43.785
C03111=1019.505,-66.061,-116.082,-24.049,21.619,-43.780
C03112=1019.508,-65.653,-116.114,-24.049,21.618,-43.774
C03113=1019.510,-65.243,-116.145,-24.050,21.617,-43.768
C03114=1019.513,-64.836,-116.175,-24.051,21.617,-43.761
C03115=1019.515,-64.427,-116.207,-24.052,21.616,-43.756
C03116=1019.518,-64.019,-116.238,-24.053,21.615,-43.750
C03117=1019.519,-63.613,-116.269,-24.053,21.615,-43.744
C03118=1019.522,-63.205,-116.300,-24.054,21.615,-43.737
C03119=1019.525,-62.799,-116.331,-24.055,21.614,-43.732
C03120=1019.527,-62.394,-116.363,-24.056,21.613,-43.726
C03121=1019.528,-61.988,-116.393,-24.057,21.612,-43.720
C03122=1019.531,-61.584,-116.424,-24.057,21.611,-43.715
C03123=1019.534,-61.180,-116.455,-24.058,21.611,-43.708
C03124=1019.535,-60.776,-116.486,-24.059,21.610,-43.702
C03125=1019.538,-60.373,-116.517,-24.060,21.610,-43.697
C03126=1019.540,-59.970,-116.548,-24.061,21.610,-43.691
C03127=1019.543,-59.568,-116.579,-24.061,21.609,-43.686
C03128=1019.544,-59.167,-116.610,-24.062,21.608,-43.680
C03129=1019.546,-58.767,-116.640,-24.063,21.608,-43.673
C03130=1019.549,-58.367,-116.672,-24.064,21.607,-43.667
C03131=1019.551,-57.967,-116.703,-24.064,21.606,-43.662
C03132=1019.553,-57.567,-116.733,-24.065,21.606,-43.656
C03133=1019.555,-57.168,-116.764,-24.066,21.605,-43.651
C03134=1019.556,-56.770,-116.795,-24.067,21.604,-43.645
C03135=1019.559,-56.372,-116.826,-24.067,21.603,-43.639
C03136=1019.560,-55.975,-116.857,-24.068,21.603,-43.632
C03137=1019.562,-55.577,-116.887,-24.069,21.602,-43.627
C03138=1019.565,-55.180,-116.918,-24.070,21.603,-43.621
C03139=1019.566,-54.783,-116.949,-24.071,21.602,-43.616
C03140=1019.568,-54.385,-116.980,-24.071,21.601,-43.610
C03141=1019.570,-53.989,-117.011,-24.072,21.600,-43.604
C03142=1019.572,-53.592,-117.042,-24.073,21.599,-43.599
C03143=1019.573,-53.195,-117.072,-24.073,21.599,-43.593
C03144=1019.575,-52.798,-117.104,-24.074,21.598,-43.588
C03145=1019.577,-52.401,-117.134,-24.075,21.598,-43.581
C03146=1019.579,-52.005,-117.165,-24.076,21.598,-43.575
C03147=1019.580,-51.608,-117.196,-24.077,21.597,-43.570
C03148=1019.582,-51.210,-117.227,-24.077,21.596,-43.564
C03149=1019.584,-50.813,-117.258,-24.078,21.595,-43.558
C03150=1019.585,-50.418,-117.289,-24.079,21.595,-43.553
C03151=1019.587,-50.020,-117.320,-24.080,21.594,-43.547
C03152=1019.588,-49.623,-117.351,-24.080,21.593,-43.542
C03153=1019.590,-49.226,-117.382,-24.081,21.592,-43.536
C03154=1019.592,-48.829,-117.413,-24.082,21.592,-43.531
C03155=1019.593,-48.431,-117.444,-24.083,21.592,-43.525
C03156=1019.594,-48.034,-117.476,-24.084,21.592,-43.518
C03157=1019.597,-47.638,-117.507,-24.084,21.591,-43.512
C03158=1019.598,-47.240,-117.538,-24.085,21.590,-43.507
C03159=1019.599,-46.843,-117.569,-24.086,21.589,-43.501
C03160=1019.600,-46.446,-117.600,-24.086,21.588,-43.496
C03161=1019.602,-46.049,-117.632,-24.087,21.589,-43.490
C03162=1019.603,-45.652,-117.663,-24.088,21.588,-43.485
C03163=1019.605,-45.254,-117.694,-24.089,21.587,-43.479
C03164=1019.606,-44.857,-117.726,-24.089,21.586,-43.473
C03165=1019.607,-44.460,-117.757,-24.090,21.585,-43.468
C03166=1019.609,-44.063,-117.788,-24.091,21.585,-43.462
C03167=1019.610,-43.666,-117.820,-24.092,21.585,-43.457
C03168=1019.612,-43.269,-117.851,-24.092,21.584,-43.451
C03169=1019.613,-42.872,-117.882,-24.093,21.584,-43.444
C03170=1019.614,-42.474,-117.913,-24.094,21.583,-43.439
C03171=1019.615,-42.077,-117.945,-24.095,21.582,-43.433
C03172=1019.617,-41.680,-117.977,-24.096,21.582,-43.427
C03173=1019.618,-41.282,-118.008,-24.096,21.582,-43.422
C03174=1019.619,-40.885,-118.039,-24.097,21.581,-43.417
C03175=1019.620,-40.488,-118.072,-24.098,21.580,-43.411
C03176=1019.621,-40.091,-118.102,-24.099,21.579,-43.405
C03177=1019.623,-39.694,-118.134,-24.099,21.579,-43.400
C03178=1019.624,-39.296,-118.166,-24.100,21.578,-43.394
C03179=1019.625,-38.899,-118.197,-24.101,21.578,-43.389
C03180=1019.626,-38.502,-118.229,-24.102,21.577,-43.383
C03181=1019.628,-38.104,-118.261,-24.102,21.576,-43.378
C03182=1019.628,-37.706,-118.293,-24.103,21.576,-43.372
C03183=1019.630,-37.309,-118.324,-24.104,21.575,-43.366
C03184=1019.630,-36.912,-118.356,-24.105,21.575,-43.361
C03185=1019.632,-36.514,-118.387,-24.105,21.574,-43.356
C03186=1019.632,-36.117,-118.419,-24.106,21.573,-43.350
C03187=1019.633,-35.720,-118.452,-24.107,21.573,-43.344
C03188=1019.635,-35.323,-118.483,-24.107,21.572,-43.339
C03189=1019.635,-34.925,-118.515,-24.108,21.572,-43.334
C03190=1019.636,-34.528,-118.547,-24.109,21.571,-43.328
C03191=1019.637,-34.131,-118.579,-24.110,21.571,-43.321
C03192=1019.638,-33.733,-118.610,-24.111,21.570,-43.315
C03193=1019.639,-33.336,-118.642,-24.111,21.570,-43.310
C03194=1019.639,-32.939,-118.674,-24.112,21.570,-43.304
C03195=1019.640,-32.541,-118.707,-24.113,21.569,-43.299
C03196=1019.641,-32.143,-118.738,-24.114,21.568,-43.293
C03197=1019.641,-31.746,-118.770,-24.114,21.567,-43.287
C03198=1019.642,-31.349,-118.802,-24.115,21.568,-43.282
C03199=1019.643,-30.952,-118.835,-24.116,21.567,-43.277
C03200=1019.644,-30.554,-118.867,-24.117,21.566,-43.271
C03201=1019.645,-30.156,-118.899,-24.117,21.565,-43.265
C03202=1019.646,-29.759,-118.931,-24.118,21.565,-43.260
C03203=1019.646,-29.361,-118.963,-24.119,21.565,-43.255
C03204=1019.647,-28.964,-118.995,-24.120,21.564,-43.249
C03205=1019.648,-28.567,-119.027,-24.120,21.563,-43.243
C03206=1019.648,-28.169,-119.059,-24.121,21.562,-43.238
C03207=1019.648,-27.772,-119.092,-24.122,21.562,-43.232
C03208=1019.649,-27.374,-119.124,-24.123,21.562,-43.227
C03209=1019.650,-26.977,-119.156,-24.123,21.561,-43.221
C03210=1019.651,-26.580,-119.188,-24.124,21.560,-43.217
C03211=1019.651,-26.182,-119.221,-24.125,21.560,-43.212
C03212=1019.651,-25.785,-119.253,-24.125,21.559,-43.206
C03213=1019.652,-25.387,-119.285,-24.126,21.558,-43.201
C03214=1019.652,-24.990,-119.317,-24.127,21.558,-43.195
C03215=1019.653,-24.592,-119.350,-24.128,21.558,-43.190
C03216=1019.653,-24.195,-119.382,-24.128,21.557,-43.184
C03217=1019.654,-23.797,-119.415,-24.129,21.556,-43.178
C03218=1019.655,-23.400,-119.447,-24.130,21.556,-43.173
C03219=1019.655,-23.002,-119.480,-24.131,21.555,-43.168
C03220=1019.655,-22.605,-119.513,-24.131,21.555,-43.162
C03221=1019.656,-22.207,-119.545,-24.132,21.554,-43.156
C03222=1019.656,-21.810,-119.578,-24.133,21.554,-43.151
C03223=1019.657,-21.412,-119.610,-24.134,21.553,-43.146
C03224=1019.656,-21.014,-119.642,-24.134,21.552,-43.140
C03225=1019.656,-20.617,-119.675,-24.135,21.553,-43.135
C03226=1019.657,-20.219,-119.707,-24.136,21.552,-43.129
C03227=1019.657,-19.822,-119.740,-24.136,21.551,-43.123
C03228=1019.657,-19.411,-119.774,-24.138,21.551,-43.116
C03229=1019.657,-19.162,-119.794,-24.138,21.550,-43.113
C03230=1019.658,-18.874,-119.817,-24.139,21.550,-43.109
C03231=1019.658,-18.562,-119.843,-24.139,21.550,-43.107
C03232=1019.658,-18.251,-119.869,-24.139,21.549,-43.105
C03233=1019.659,-17.963,-119.893,-24.139,21.549,-43.101
C03234=1019.659,-17.715,-119.912,-24.140,21.548,-43.098
C03235=1019.659,-17.304,-119.947,-24.141,21.547,-43.090
C03236=1019.659,-16.907,-119.980,-24.142,21.548,-43.085
C03237=1019.659,-16.509,-120.012,-24.142,21.547,-43.079
C03238=1019.658,-16.110,-120.045,-24.143,21.546,-43.074
C03239=1019.659,-15.710,-120.078,-24.144,21.546,-43.068
C03240=1019.659,-15.310,-120.111,-24.145,21.545,-43.063
C03241=1019.659,-14.907,-120.144,-24.145,21.545,-43.057
C03242=1019.659,-14.502,-120.178,-24.146,21.544,-43.052
C03243=1019.659,-14.093,-120.212,-24.147,21.544,-43.046
C03244=1019.659,-13.681,-120.247,-24.148,21.543,-43.041
C03245=1019.659,-13.267,-120.280,-24.148,21.543,-43.035
C03246=1019.659,-12.849,-120.315,-24.149,21.542,-43.029
C03247=1019.659,-12.430,-120.350,-24.150,21.542,-43.024
C03248=1019.659,-12.219,-120.368,-24.150,21.541,-43.022
C03249=1019.659,-12.007,-120.385,-24.151,21.541,-43.019
C03250=1019.659,-11.796,-120.403,-24.151,21.540,-43.016
C03251=1019.658,-11.584,-120.420,-24.151,21.540,-43.013
C03252=1019.659,-11.371,-120.437,-24.152,21.540,-43.011
C03253=1019.659,-11.157,-120.456,-24.152,21.540,-43.007
C03254=1019.658,-10.943,-120.473,-24.152,21.539,-43.006
C03255=1019.658,-10.730,-120.491,-24.153,21.539,-43.002
C03256=1019.659,-10.515,-120.509,-24.153,21.539,-42.998
C03257=1019.658,-10.300,-120.527,-24.154,21.538,-42.996
C03258=1019.659,-10.084,-120.544,-24.154,21.539,-42.993
C03259=1019.659,-9.869,-120.563,-24.154,21.538,-42.991
C03260=1019.658,-9.653,-120.580,-24.155,21.538,-42.987
C03261=1019.658,-9.437,-120.599,-24.155,21.538,-42.985
C03262=1019.659,-9.221,-120.617,-24.156,21.537,-42.982
C03263=1019.658,-9.005,-120.635,-24.156,21.537,-42.980
C03264=1019.658,-8.788,-120.653,-24.156,21.536,-42.976
C03265=1019.658,-8.571,-120.671,-24.157,21.537,-42.973
C03266=1019.658,-8.354,-120.689,-24.157,21.536,-42.971
C03267=1019.658,-8.138,-120.707,-24.158,21.536,-42.967
C03268=1019.657,-7.921,-120.726,-24.158,21.536,-42.965
C03269=1019.657,-7.704,-120.743,-24.158,21.535,-42.961
C03270=1019.657,-7.486,-120.761,-24.159,21.535,-42.959
C03271=1019.657,-7.266,-120.780,-24.159,21.534,-42.956
C03272=1019.657,-7.046,-120.798,-24.160,21.535,-42.952
C03273=1019.657,-6.824,-120.817,-24.160,21.534,-42.950
C03274=1019.657,-6.602,-120.836,-24.160,21.534,-42.947
C03275=1019.656,-6.379,-120.854,-24.161,21.533,-42.944
C03276=1019.656,-6.155,-120.873,-24.161,21.533,-42.941
C03277=1019.656,-5.930,-120.891,-24.161,21.533,-42.939
C03278=1019.656,-5.707,-120.910,-24.162,21.533,-42.935
C03279=1019.656,-5.482,-120.929,-24.162,21.532,-42.934
C03280=1019.655,-5.259,-120.948,-24.163,21.532,-42.930
C03281=1019.655,-5.036,-120.967,-24.163,21.532,-42.927
C03282=1019.655,-4.815,-120.985,-24.163,21.532,-42.925
C03283=1019.655,-4.595,-121.003,-24.164,21.531,-42.921
C03284=1019.655,-4.377,-121.022,-24.164,21.531,-42.919
C03285=1019.654,-4.160,-121.040,-24.165,21.531,-42.915
C03286=1019.654,-3.944,-121.059,-24.165,21.530,-42.913
C03287=1019.654,-3.731,-121.077,-24.165,21.530,-42.910
C03288=1019.654,-3.518,-121.094,-24.166,21.530,-42.908
C03289=1019.654,-3.307,-121.112,-24.166,21.530,-42.904
C03290=1019.653,-2.886,-121.148,-24.167,21.529,-42.899
C03291=1019.652,-2.467,-121.183,-24.168,21.529,-42.893
C03292=1019.652,-2.049,-121.218,-24.169,21.529,-42.888
C03293=1019.652,-1.634,-121.253,-24.169,21.528,-42.882
C03294=1019.651,-1.221,-121.287,-24.170,21.527,-42.877
C03295=1019.650,-0.812,-121.323,-24.171,21.527,-42.872
C03296=1019.650,-0.403,-121.356,-24.171,21.526,-42.867
C03297=1019.649,0.001,-121.391,-24.172,21.525,-42.862
C03298=1019.649,0.405,-121.425,-24.173,21.525,-42.857
C03299=1019.648,0.807,-121.459,-24.173,21.525,-42.851
C03300=1019.648,1.206,-121.492,-24.174,21.525,-42.846
C03301=1019.647,1.605,-121.526,-24.175,21.523,-42.841
C03302=1019.647,2.004,-121.560,-24.175,21.524,-42.836
C03303=1019.646,2.390,-121.593,-24.176,21.523,-42.833
C03304=1019.645,2.742,-121.622,-24.177,21.522,-42.827
C03305=1019.645,3.065,-121.650,-24.177,21.522,-42.823
C03306=1019.644,3.378,-121.676,-24.178,21.521,-42.817
C03307=1019.643,3.707,-121.705,-24.179,21.521,-42.812
C03308=1019.643,4.066,-121.735,-24.179,21.521,-42.809
C03309=1019.642,4.455,-121.769,-24.180,21.520,-42.805
C03310=1019.641,4.851,-121.802,-24.180,21.519,-42.799
C03311=1019.641,5.246,-121.836,-24.181,21.520,-42.794
C03312=1019.640,5.641,-121.869,-24.182,21.519,-42.790
C03313=1019.640,6.036,-121.903,-24.182,21.518,-42.785
C03314=1019.639,6.429,-121.937,-24.183,21.519,-42.779
C03315=1019.637,6.822,-121.970,-24.184,21.517,-42.775
C03316=1019.637,7.215,-122.003,-24.185,21.517,-42.770
C03317=1019.636,7.605,-122.037,-24.185,21.517,-42.764
C03318=1019.635,7.993,-122.070,-24.186,21.516,-42.761
C03319=1019.634,8.377,-122.102,-24.187,21.516,-42.755
C03320=1019.634,8.758,-122.135,-24.187,21.515,-42.751
C03321=1019.632,9.136,-122.168,-24.188,21.515,-42.746
C03322=1019.631,9.512,-122.199,-24.189,21.514,-42.740
C03323=1019.630,9.888,-122.232,-24.189,21.514,-42.737
C03324=1019.630,10.264,-122.264,-24.190,21.513,-42.731
C03325=1019.629,10.643,-122.297,-24.191,21.513,-42.726
C03326=1019.628,11.023,-122.329,-24.191,21.513,-42.722
C03327=1019.627,11.406,-122.361,-24.192,21.512,-42.716
C03328=1019.625,11.792,-122.395,-24.192,21.511,-42.713
C03329=1019.625,12.178,-122.428,-24.193,21.512,-42.707
C03330=1019.624,12.565,-122.462,-24.193,21.510,-42.703
C03331=1019.623,12.951,-122.495,-24.194,21.510,-42.698
C03332=1019.622,13.338,-122.528,-24.195,21.511,-42.693
C03333=1019.621,13.725,-122.561,-24.196,21.509,-42.689
C03334=1019.620,14.112,-122.594,-24.196,21.509,-42.683
C03335=1019.619,14.500,-122.628,-24.197,21.509,-42.680
C03336=1019.617,14.889,-122.662,-24.198,21.508,-42.674
C03337=1019.617,15.277,-122.695,-24.198,21.508,-42.670
C03338=1019.615,15.667,-122.728,-24.199,21.507,-42.665
C03339=1019.614,16.056,-122.762,-24.200,21.507,-42.659
C03340=1019.612,16.448,-122.796,-24.200,21.506,-42.656
C03341=1019.612,16.840,-122.829,-24.201,21.506,-42.650
C03342=1019.610,17.232,-122.864,-24.201,21.505,-42.646
C03343=1019.609,17.626,-122.898,-24.202,21.505,-42.641
C03344=1019.608,18.020,-122.932,-24.203,21.505,-42.635
C03345=1019.606,18.415,-122.966,-24.203,21.504,-42.632
C03346=1019.605,18.810,-123.001,-24.204,21.503,-42.626
C03347=1019.604,19.207,-123.034,-24.205,21.503,-42.622
C03348=1019.603,19.604,-123.069,-24.205,21.503,-42.617
C03349=1019.602,19.815,-123.087,-24.206,21.503,-42.613
C03350=1019.601,20.052,-123.108,-24.206,21.502,-42.610
C03351=1019.600,20.318,-123.131,-24.207,21.503,-42.606
C03352=1019.600,20.604,-123.156,-24.207,21.501,-42.604
C03353=1019.599,20.901,-123.182,-24.207,21.501,-42.602
C03354=1019.597,21.193,-123.207,-24.208,21.502,-42.599
C03355=1019.596,21.465,-123.231,-24.208,21.501,-42.597
C03356=1019.596,21.709,-123.252,-24.209,21.501,-42.593
C03357=1019.594,22.123,-123.288,-24.210,21.501,-42.586
C03358=1019.593,22.498,-123.321,-24.210,21.500,-42.584
C03359=1019.592,22.820,-123.349,-24.211,21.500,-42.580
C03360=1019.590,23.086,-123.372,-24.211,21.500,-42.577
C03361=1019.589,23.318,-123.393,-24.211,21.499,-42.573
C03362=1019.589,23.553,-123.412,-24.212,21.498,-42.567
C03363=1019.588,23.824,-123.436,-24.213,21.498,-42.564
C03364=1019.587,24.154,-123.465,-24.213,21.498,-42.562
C03365=1019.585,24.538,-123.498,-24.213,21.497,-42.558
C03366=1019.584,24.937,-123.533,-24.214,21.497,-42.553
C03367=1019.582,25.336,-123.568,-24.215,21.497,-42.549
C03368=1019.580,25.735,-123.603,-24.215,21.496,-42.543
C03369=1019.579,26.134,-123.638,-24.216,21.496,-42.540
C03370=1019.578,26.534,-123.673,-24.217,21.496,-42.534
C03371=1019.576,26.934,-123.708,-24.218,21.495,-42.529
C03372=1019.575,27.333,-123.743,-24.218,21.494,-42.525
C03373=1019.572,27.732,-123.778,-24.219,21.495,-42.520
C03374=1019.571,28.131,-123.813,-24.219,21.493,-42.516
C03375=1019.569,28.531,-123.848,-24.220,21.493,-42.510
C03376=1019.567,28.931,-123.883,-24.221,21.493,-42.507
C03377=1019.566,29.330,-123.918,-24.221,21.492,-42.501
C03378=1019.564,29.730,-123.953,-24.222,21.492,-42.497
C03379=1019.562,30.129,-123.988,-24.223,21.492,-42.492
C03380=1019.561,30.528,-124.023,-24.223,21.491,-42.488
C03381=1019.558,30.928,-124.059,-24.224,21.491,-42.483
C03382=1019.557,31.328,-124.094,-24.224,21.490,-42.479
C03383=1019.555,31.727,-124.130,-24.225,21.490,-42.474
C03384=1019.553,32.127,-124.164,-24.226,21.489,-42.469
C03385=1019.552,32.527,-124.199,-24.226,21.489,-42.464
C03386=1019.550,32.927,-124.235,-24.227,21.489,-42.461
C03387=1019.548,33.326,-124.270,-24.228,21.489,-42.455
C03388=1019.546,33.725,-124.305,-24.228,21.487,-42.451
C03389=1019.544,34.126,-124.341,-24.229,21.488,-42.446
C03390=1019.543,34.525,-124.376,-24.229,21.487,-42.442
C03391=1019.540,34.925,-124.411,-24.230,21.486,-42.437
C03392=1019.539,35.325,-124.446,-24.231,21.486,-42.433
C03393=1019.537,35.725,-124.482,-24.231,21.486,-42.428
C03394=1019.534,36.124,-124.517,-24.232,21.486,-42.424
C03395=1019.533,36.524,-124.553,-24.233,21.485,-42.418
C03396=1019.531,36.924,-124.588,-24.233,21.484,-42.414
C03397=1019.529,37.324,-124.623,-24.234,21.485,-42.409
C03398=1019.527,37.724,-124.659,-24.235,21.484,-42.405
C03399=1019.524,38.123,-124.694,-24.235,21.483,-42.400
C03400=1019.523,38.524,-124.730,-24.236,21.483,-42.396
C03401=1019.520,38.923,-124.766,-24.237,21.483,-42.391
C03402=1019.519,39.324,-124.801,-24.237,21.483,-42.387
C03403=1019.517,39.723,-124.836,-24.238,21.482,-42.383
C03404=1019.514,40.123,-124.871,-24.238,21.481,-42.378
C03405=1019.513,40.523,-124.907,-24.239,21.481,-42.374
C03406=1019.510,40.923,-124.943,-24.240,21.481,-42.369
C03407=1019.508,41.323,-124.979,-24.240,21.481,-42.365
C03408=1019.506,41.723,-125.015,-24.241,21.480,-42.359
C03409=1019.504,42.123,-125.050,-24.241,21.479,-42.356
C03410=1019.501,42.523,-125.085,-24.242,21.479,-42.352
C03411=1019.499,42.923,-125.121,-24.243,21.479,-42.347
C03412=1019.497,43.323,-125.157,-24.243,21.479,-42.343
C03413=1019.495,43.722,-125.192,-24.244,21.479,-42.338
C03414=1019.492,44.123,-125.229,-24.244,21.477,-42.333
C03415=1019.490,44.523,-125.264,-24.245,21.477,-42.330
C03416=1019.488,44.923,-125.299,-24.246,21.477,-42.325
C03417=1019.486,45.323,-125.335,-24.246,21.477,-42.321
C03418=1019.483,45.724,-125.371,-24.247,21.477,-42.316
C03419=1019.481,46.123,-125.407,-24.247,21.475,-42.311
C03420=1019.479,46.523,-125.443,-24.248,21.475,-42.308
C03421=1019.476,46.923,-125.479,-24.249,21.475,-42.302
C03422=1019.474,47.323,-125.515,-24.249,21.475,-42.299
C03423=1019.471,47.724,-125.550,-24.250,21.474,-42.295
C03424=1019.469,48.124,-125.586,-24.251,21.474,-42.290
C03425=1019.467,48.524,-125.622,-24.251,21.474,-42.286
C03426=1019.464,48.924,-125.658,-24.251,21.472,-42.282
C03427=1019.462,49.324,-125.694,-24.252,21.473,-42.277
C03428=1019.460,49.724,-125.730,-24.253,21.472,-42.273
C03429=1019.457,50.124,-125.766,-24.254,21.472,-42.268
C03430=1019.455,50.524,-125.802,-24.254,21.472,-42.264
C03431=1019.451,50.925,-125.838,-24.255,21.471,-42.260
C03432=1019.450,51.325,-125.873,-24.255,21.471,-42.255
C03433=1019.447,51.725,-125.910,-24.256,21.471,-42.251
C03434=1019.444,52.125,-125.946,-24.256,21.470,-42.247
C03435=1019.442,52.525,-125.982,-24.257,21.469,-42.243
C03436=1019.439,52.926,-126.018,-24.258,21.469,-42.238
C03437=1019.436,53.325,-126.054,-24.258,21.469,-42.234
C03438=1019.434,53.726,-126.091,-24.259,21.468,-42.230
C03439=1019.432,54.126,-126.127,-24.259,21.468,-42.225
C03440=1019.429,54.526,-126.163,-24.260,21.468,-42.221
C03441=1019.427,54.927,-126.199,-24.260,21.468,-42.218
C03442=1019.423,55.327,-126.235,-24.261,21.468,-42.212
C03443=1019.421,55.728,-126.271,-24.262,21.467,-42.209
C03444=1019.418,56.127,-126.307,-24.262,21.467,-42.205
C03445=1019.416,56.528,-126.343,-24.263,21.465,-42.201
C03446=1019.413,56.928,-126.379,-24.264,21.466,-42.196
C03447=1019.410,57.327,-126.415,-24.264,21.465,-42.192
C03448=1019.407,57.728,-126.452,-24.264,21.465,-42.188
C03449=1019.404,58.128,-126.488,-24.265,21.465,-42.183
C03450=1019.402,58.528,-126.524,-24.266,21.464,-42.179
C03451=1019.399,58.928,-126.561,-24.266,21.464,-42.175
C03452=1019.396,59.329,-126.597,-24.267,21.463,-42.172
C03453=1019.393,59.729,-126.633,-24.268,21.464,-42.166
C03454=1019.391,60.129,-126.670,-24.268,21.463,-42.163
C03455=1019.388,60.529,-126.706,-24.269,21.463,-42.159
C03456=1019.385,60.930,-126.742,-24.269,21.462,-42.155
C03457=1019.381,61.330,-126.779,-24.270,21.462,-42.150
C03458=1019.379,61.730,-126.815,-24.270,21.462,-42.146
C03459=1019.376,62.130,-126.852,-24.271,21.461,-42.142
C03460=1019.373,62.530,-126.888,-24.271,21.461,-42.139
C03461=1019.370,62.950,-126.926,-24.272,21.460,-42.133
C03462=1019.368,63.204,-126.949,-24.272,21.460,-42.131
C03463=1019.366,63.471,-126.973,-24.273,21.460,-42.129
C03464=1019.364,63.721,-126.996,-24.273,21.459,-42.127
C03465=1019.363,63.937,-127.016,-24.274,21.460,-42.124
C03466=1019.361,64.144,-127.035,-24.274,21.460,-42.122
C03467=1019.360,64.363,-127.055,-24.274,21.459,-42.120
C03468=1019.358,64.592,-127.076,-24.274,21.459,-42.116
C03469=1019.356,64.828,-127.097,-24.275,21.459,-42.115
C03470=1019.355,65.064,-127.119,-24.275,21.458,-42.113
C03471=1019.353,65.294,-127.140,-24.275,21.458,-42.111
C03472=1019.351,65.515,-127.160,-24.276,21.459,-42.108
C03473=1019.349,65.728,-127.180,-24.276,21.458,-42.106
C03474=1019.346,66.136,-127.216,-24.277,21.458,-42.102
C03475=1019.343,66.534,-127.253,-24.277,21.457,-42.098
C03476=1019.340,66.935,-127.290,-24.278,21.457,-42.094
C03477=1019.337,67.337,-127.326,-24.278,21.457,-42.089
C03478=1019.334,67.741,-127.364,-24.279,21.457,-42.085
C03479=1019.330,68.145,-127.400,-24.279,21.456,-42.082
C03480=1019.327,68.551,-127.438,-24.280,21.456,-42.078
C03481=1019.324,68.959,-127.475,-24.280,21.455,-42.074
C03482=1019.321,69.367,-127.513,-24.281,21.455,-42.069
C03483=1019.318,69.777,-127.550,-24.282,21.455,-42.065
C03484=1019.314,70.189,-127.588,-24.282,21.454,-42.061
C03485=1019.311,70.600,-127.625,-24.283,21.454,-42.058
C03486=1019.308,71.011,-127.663,-24.283,21.453,-42.054
C03487=1019.304,71.422,-127.701,-24.284,21.454,-42.049
C03488=1019.301,71.834,-127.739,-24.285,21.453,-42.045
C03489=1019.298,72.246,-127.776,-24.285,21.453,-42.041
C03490=1019.295,72.659,-127.814,-24.285,21.452,-42.037
C03491=1019.291,73.074,-127.853,-24.286,21.452,-42.034
C03492=1019.288,73.492,-127.891,-24.287,21.452,-42.028
C03493=1019.284,73.912,-127.929,-24.287,21.452,-42.025
C03494=1019.282,74.124,-127.949,-24.288,21.451,-42.023
C03495=1019.281,74.336,-127.969,-24.288,21.451,-42.021
C03496=1019.279,74.548,-127.988,-24.288,21.451,-42.019
C03497=1019.277,74.762,-128.007,-24.288,21.451,-42.017
C03498=1019.275,74.975,-128.027,-24.289,21.450,-42.015
C03499=1019.273,75.189,-128.046,-24.289,21.451,-42.012
C03500=1019.271,75.402,-128.067,-24.289,21.451,-42.010
C03501=1019.269,75.615,-128.086,-24.290,21.450,-42.008
C03502=1019.266,76.035,-128.125,-24.290,21.450,-42.004
C03503=1019.262,76.446,-128.163,-24.291,21.449,-42.001
C03504=1019.259,76.849,-128.200,-24.291,21.449,-41.997
C03505=1019.256,77.243,-128.236,-24.292,21.449,-41.994
C03506=1019.252,77.632,-128.272,-24.292,21.448,-41.989
C03507=1019.249,78.018,-128.307,-24.293,21.447,-41.986
C03508=1019.246,78.404,-128.343,-24.293,21.448,-41.980
C03509=1019.242,78.795,-128.379,-24.294,21.447,-41.977
C03510=1019.239,79.192,-128.416,-24.294,21.447,-41.973
C03511=1019.235,79.597,-128.453,-24.295,21.447,-41.970
C03512=1019.231,80.012,-128.492,-24.296,21.447,-41.966
C03513=1019.230,80.222,-128.511,-24.296,21.446,-41.964
C03514=1019.227,80.434,-128.530,-24.296,21.446,-41.962
C03515=1019.226,80.647,-128.550,-24.296,21.446,-41.960
C03516=1019.224,80.859,-128.569,-24.297,21.446,-41.958
C03517=1019.221,81.072,-128.590,-24.297,21.445,-41.956
C03518=1019.219,81.285,-128.609,-24.297,21.445,-41.955
C03519=1019.218,81.498,-128.629,-24.297,21.445,-41.953
C03520=1019.216,81.709,-128.649,-24.298,21.445,-41.951
C03521=1019.214,81.922,-128.668,-24.298,21.445,-41.949
C03522=1019.213,82.133,-128.688,-24.298,21.444,-41.947
C03523=1019.210,82.345,-128.707,-24.299,21.445,-41.944
C03524=1019.208,82.556,-128.727,-24.299,21.444,-41.942
C03525=1019.206,82.768,-128.747,-24.299,21.444,-41.940
C03526=1019.204,82.977,-128.766,-24.299,21.444,-41.938
C03527=1019.201,83.398,-128.806,-24.300,21.444,-41.935
C03528=1019.197,83.817,-128.844,-24.300,21.444,-41.931
C03529=1019.192,84.234,-128.883,-24.301,21.443,-41.927
C03530=1019.188,84.650,-128.921,-24.301,21.443,-41.923
C03531=1019.185,85.064,-128.960,-24.302,21.443,-41.920
C03532=1019.181,85.477,-128.998,-24.302,21.442,-41.916
C03533=1019.178,85.887,-129.036,-24.303,21.442,-41.912
C03534=1019.174,86.296,-129.074,-24.303,21.441,-41.908
C03535=1019.169,86.703,-129.112,-24.304,21.442,-41.905
C03536=1019.165,87.110,-129.150,-24.304,21.441,-41.901
C03537=1019.162,87.513,-129.187,-24.305,21.441,-41.898
C03538=1019.158,87.908,-129.224,-24.305,21.440,-41.894
C03539=1019.154,88.297,-129.260,-24.306,21.440,-41.890
C03540=1019.150,88.680,-129.296,-24.307,21.440,-41.887
C03541=1019.147,89.062,-129.331,-24.307,21.440,-41.883
C03542=1019.142,89.449,-129.368,-24.308,21.439,-41.879
C03543=1019.139,89.842,-129.404,-24.308,21.439,-41.875
C03544=1019.135,90.240,-129.441,-24.309,21.439,-41.872
C03545=1019.131,90.639,-129.478,-24.309,21.439,-41.868
C03546=1019.127,91.039,-129.515,-24.310,21.438,-41.865
C03547=1019.123,91.438,-129.552,-24.310,21.438,-41.861
C03548=1019.120,91.838,-129.590,-24.311,21.438,-41.857
C03549=1019.115,92.237,-129.627,-24.311,21.438,-41.854
C03550=1019.111,92.636,-129.664,-24.312,21.437,-41.850
C03551=1019.107,93.035,-129.701,-24.312,21.437,-41.846
C03552=1019.103,93.434,-129.739,-24.312,21.437,-41.844
C03553=1019.099,93.833,-129.776,-24.313,21.436,-41.841
C03554=1019.095,94.232,-129.813,-24.313,21.436,-41.837
C03555=1019.091,94.632,-129.851,-24.314,21.435,-41.833
C03556=1019.087,95.030,-129.888,-24.315,21.436,-41.830
C03557=1019.083,95.429,-129.926,-24.315,21.435,-41.826
C03558=1019.079,95.828,-129.963,-24.316,21.435,-41.822
C03559=1019.075,96.226,-130.000,-24.316,21.435,-41.819
C03560=1019.070,96.625,-130.038,-24.317,21.435,-41.815
C03561=1019.066,97.025,-130.075,-24.317,21.434,-41.811
C03562=1019.062,97.424,-130.112,-24.318,21.434,-41.808
C03563=1019.058,97.823,-130.149,-24.318,21.433,-41.806
C03564=1019.053,98.222,-130.187,-24.318,21.433,-41.802
C03565=1019.050,98.620,-130.225,-24.319,21.432,-41.798
C03566=1019.046,99.019,-130.262,-24.319,21.433,-41.795
C03567=1019.041,99.418,-130.299,-24.320,21.432,-41.791
C03568=1019.037,99.817,-130.336,-24.320,21.432,-41.787
C03569=1019.033,100.216,-130.374,-24.321,21.432,-41.784
C03570=1019.028,100.614,-130.412,-24.322,21.432,-41.780
C03571=1019.024,101.013,-130.449,-24.322,21.431,-41.778
C03572=1019.019,101.412,-130.487,-24.322,21.431,-41.775
C03573=1019.015,101.811,-130.524,-24.323,21.431,-41.771
C03574=1019.011,102.210,-130.561,-24.323,21.430,-41.767
C03575=1019.006,102.608,-130.599,-24.324,21.430,-41.763
C03576=1019.002,103.007,-130.636,-24.324,21.430,-41.760
C03577=1018.997,103.406,-130.674,-24.325,21.430,-41.756
